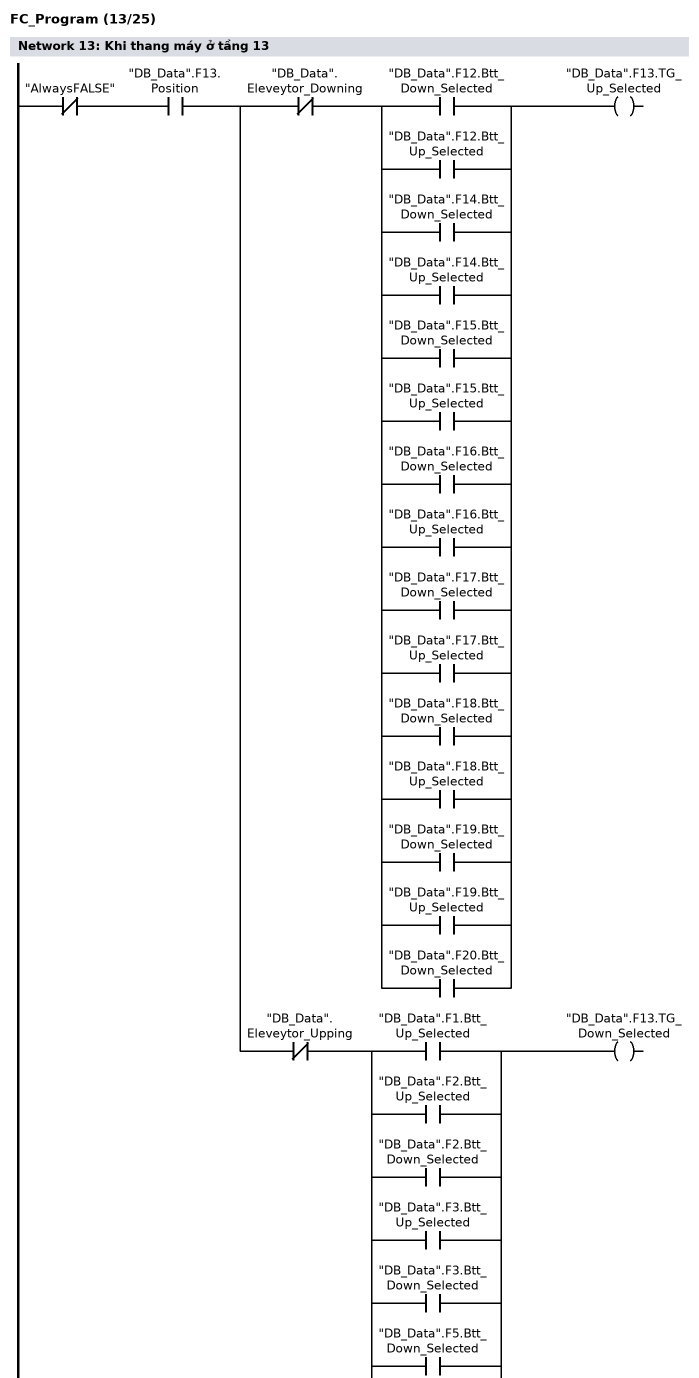
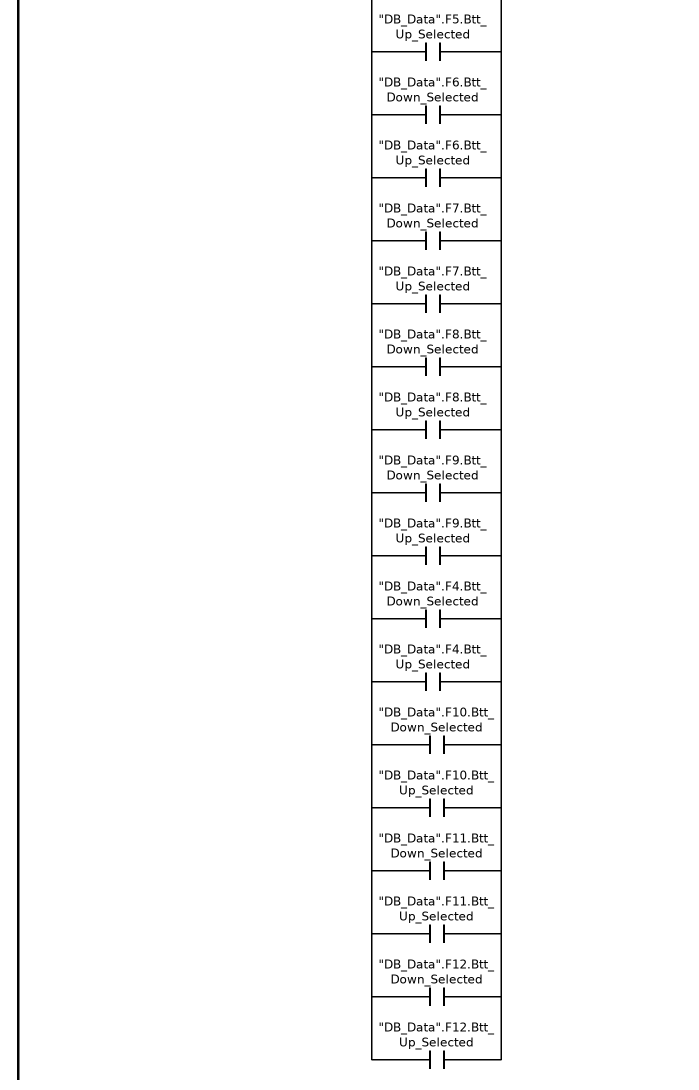
   RUNG wire#powerrail
      I_Contact( "AlwaysFALSE" )
      Contact( "DB_Data".F13.Position )
      wire#w1
      I_Contact( "DB_Data".Eleveytor_Downing )
      wire#w2
      Contact( "DB_Data".F12.Btt_Down_Selected )
      wire#w3
      Coil( "DB_Data".F13.TG_Up_Selected )
   END_RUNG
   RUNG wire#w2
      Contact( "DB_Data".F12.Btt_Up_Selected )
   END_RUNG wire#w3
   RUNG wire#w2
      Contact( "DB_Data".F14.Btt_Down_Selected )
   END_RUNG wire#w3
   RUNG wire#w2
      Contact( "DB_Data".F14.Btt_Up_Selected )
   END_RUNG wire#w3
   RUNG wire#w2
      Contact( "DB_Data".F15.Btt_Down_Selected )
   END_RUNG wire#w3
   RUNG wire#w2
      Contact( "DB_Data".F15.Btt_Up_Selected )
   END_RUNG wire#w3
   RUNG wire#w2
      Contact( "DB_Data".F16.Btt_Down_Selected )
   END_RUNG wire#w3
   RUNG wire#w2
      Contact( "DB_Data".F16.Btt_Up_Selected )
   END_RUNG wire#w3
   RUNG wire#w2
      Contact( "DB_Data".F17.Btt_Down_Selected )
   END_RUNG wire#w3
   RUNG wire#w2
      Contact( "DB_Data".F17.Btt_Up_Selected )
   END_RUNG wire#w3
   RUNG wire#w2
      Contact( "DB_Data".F18.Btt_Down_Selected )
   END_RUNG wire#w3
   RUNG wire#w2
      Contact( "DB_Data".F18.Btt_Up_Selected )
   END_RUNG wire#w3
   RUNG wire#w2
      Contact( "DB_Data".F19.Btt_Down_Selected )
   END_RUNG wire#w3
   RUNG wire#w2
      Contact( "DB_Data".F19.Btt_Up_Selected )
   END_RUNG wire#w3
   RUNG wire#w2
      Contact( "DB_Data".F20.Btt_Down_Selected )
   END_RUNG wire#w3
   RUNG wire#w1
      I_Contact( "DB_Data".Eleveytor_Upping )
      wire#w4
      Contact( "DB_Data".F1.Btt_Up_Selected )
      wire#w5
      Coil( "DB_Data".F13.TG_Down_Selected )
   END_RUNG
   RUNG wire#w4
      Contact( "DB_Data".F2.Btt_Up_Selected )
   END_RUNG wire#w5
   RUNG wire#w4
      Contact( "DB_Data".F2.Btt_Down_Selected )
   END_RUNG wire#w5
   RUNG wire#w4
      Contact( "DB_Data".F3.Btt_Up_Selected )
   END_RUNG wire#w5
   RUNG wire#w4
      Contact( "DB_Data".F3.Btt_Down_Selected )
   END_RUNG wire#w5
   RUNG wire#w4
      Contact( "DB_Data".F5.Btt_Down_Selected )
   END_RUNG wire#w5
   RUNG wire#w4
      Contact( "DB_Data".F5.Btt_Up_Selected )
   END_RUNG wire#w5
   RUNG wire#w4
      Contact( "DB_Data".F6.Btt_Down_Selected )
   END_RUNG wire#w5
   RUNG wire#w4
      Contact( "DB_Data".F6.Btt_Up_Selected )
   END_RUNG wire#w5
   RUNG wire#w4
      Contact( "DB_Data".F7.Btt_Down_Selected )
   END_RUNG wire#w5
   RUNG wire#w4
      Contact( "DB_Data".F7.Btt_Up_Selected )
   END_RUNG wire#w5
   RUNG wire#w4
      Contact( "DB_Data".F8.Btt_Down_Selected )
   END_RUNG wire#w5
   RUNG wire#w4
      Contact( "DB_Data".F8.Btt_Up_Selected )
   END_RUNG wire#w5
   RUNG wire#w4
      Contact( "DB_Data".F9.Btt_Down_Selected )
   END_RUNG wire#w5
   RUNG wire#w4
      Contact( "DB_Data".F9.Btt_Up_Selected )
   END_RUNG wire#w5
   RUNG wire#w4
      Contact( "DB_Data".F4.Btt_Down_Selected )
   END_RUNG wire#w5
   RUNG wire#w4
      Contact( "DB_Data".F4.Btt_Up_Selected )
   END_RUNG wire#w5
   RUNG wire#w4
      Contact( "DB_Data".F10.Btt_Down_Selected )
   END_RUNG wire#w5
   RUNG wire#w4
      Contact( "DB_Data".F10.Btt_Up_Selected )
   END_RUNG wire#w5
   RUNG wire#w4
      Contact( "DB_Data".F11.Btt_Down_Selected )
   END_RUNG wire#w5
   RUNG wire#w4
      Contact( "DB_Data".F11.Btt_Up_Selected )
   END_RUNG wire#w5
   RUNG wire#w4
      Contact( "DB_Data".F12.Btt_Down_Selected )
   END_RUNG wire#w5
   RUNG wire#w4
      Contact( "DB_Data".F12.Btt_Up_Selected )
   END_RUNG wire#w5
   // the same network as SCL:
   #_w1 := NOT "AlwaysFALSE" AND "DB_Data".F13.Position;
   "DB_Data".F13.TG_Up_Selected := #_w1 AND NOT "DB_Data".Eleveytor_Downing AND ("DB_Data".F12.Btt_Down_Selected OR "DB_Data".F12.Btt_Up_Selected OR "DB_Data".F14.Btt_Down_Selected OR "DB_Data".F14.Btt_Up_Selected OR "DB_Data".F15.Btt_Down_Selected OR "DB_Data".F15.Btt_Up_Selected OR "DB_Data".F16.Btt_Down_Selected OR "DB_Data".F16.Btt_Up_Selected OR "DB_Data".F17.Btt_Down_Selected OR "DB_Data".F17.Btt_Up_Selected OR "DB_Data".F18.Btt_Down_Selected OR "DB_Data".F18.Btt_Up_Selected OR "DB_Data".F19.Btt_Down_Selected OR "DB_Data".F19.Btt_Up_Selected OR "DB_Data".F20.Btt_Down_Selected);
   "DB_Data".F13.TG_Down_Selected := #_w1 AND NOT "DB_Data".Eleveytor_Upping AND ("DB_Data".F1.Btt_Up_Selected OR "DB_Data".F2.Btt_Up_Selected OR "DB_Data".F2.Btt_Down_Selected OR "DB_Data".F3.Btt_Up_Selected OR "DB_Data".F3.Btt_Down_Selected OR "DB_Data".F5.Btt_Down_Selected OR "DB_Data".F5.Btt_Up_Selected OR "DB_Data".F6.Btt_Down_Selected OR "DB_Data".F6.Btt_Up_Selected OR "DB_Data".F7.Btt_Down_Selected OR "DB_Data".F7.Btt_Up_Selected OR "DB_Data".F8.Btt_Down_Selected OR "DB_Data".F8.Btt_Up_Selected OR "DB_Data".F9.Btt_Down_Selected OR "DB_Data".F9.Btt_Up_Selected OR "DB_Data".F4.Btt_Down_Selected OR "DB_Data".F4.Btt_Up_Selected OR "DB_Data".F10.Btt_Down_Selected OR "DB_Data".F10.Btt_Up_Selected OR "DB_Data".F11.Btt_Down_Selected OR "DB_Data".F11.Btt_Up_Selected OR "DB_Data".F12.Btt_Down_Selected OR "DB_Data".F12.Btt_Up_Selected);
END_REGION

REGION Network 14: Khi thang máy ở tầng 14
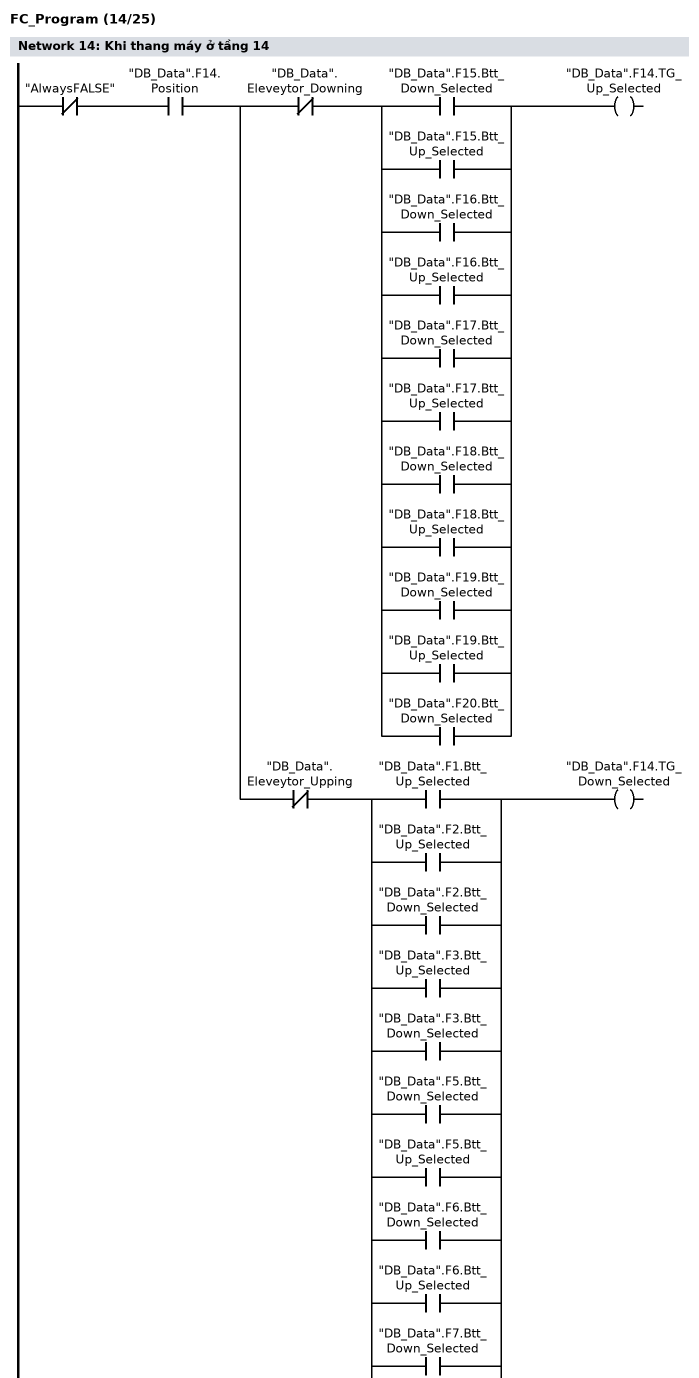
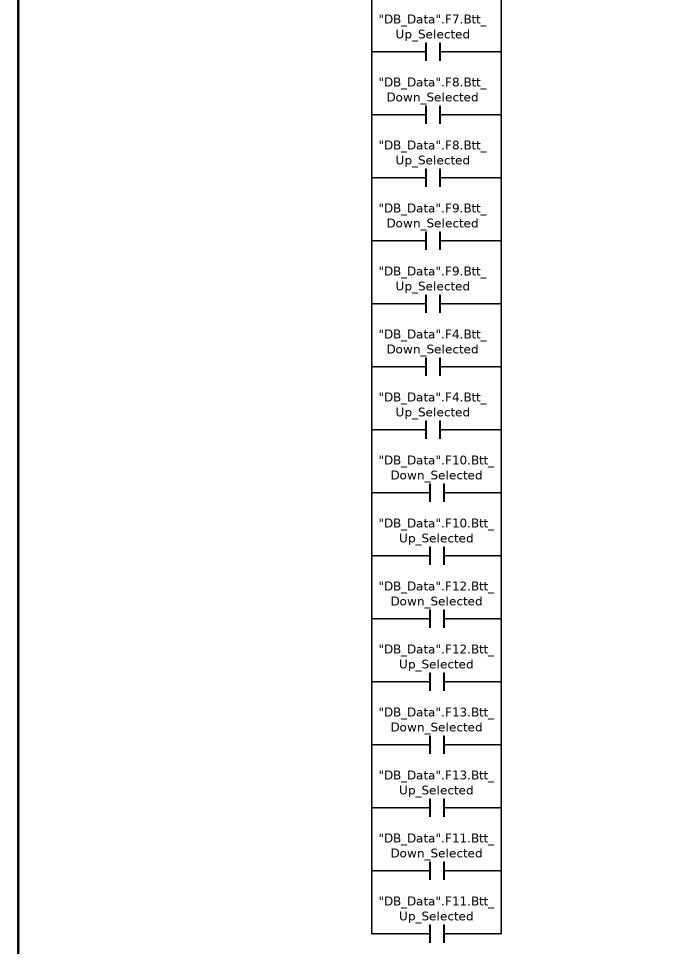
   RUNG wire#powerrail
      I_Contact( "AlwaysFALSE" )
      Contact( "DB_Data".F14.Position )
      wire#w1
      I_Contact( "DB_Data".Eleveytor_Downing )
      wire#w2
      Contact( "DB_Data".F15.Btt_Down_Selected )
      wire#w3
      Coil( "DB_Data".F14.TG_Up_Selected )
   END_RUNG
   RUNG wire#w2
      Contact( "DB_Data".F15.Btt_Up_Selected )
   END_RUNG wire#w3
   RUNG wire#w2
      Contact( "DB_Data".F16.Btt_Down_Selected )
   END_RUNG wire#w3
   RUNG wire#w2
      Contact( "DB_Data".F16.Btt_Up_Selected )
   END_RUNG wire#w3
   RUNG wire#w2
      Contact( "DB_Data".F17.Btt_Down_Selected )
   END_RUNG wire#w3
   RUNG wire#w2
      Contact( "DB_Data".F17.Btt_Up_Selected )
   END_RUNG wire#w3
   RUNG wire#w2
      Contact( "DB_Data".F18.Btt_Down_Selected )
   END_RUNG wire#w3
   RUNG wire#w2
      Contact( "DB_Data".F18.Btt_Up_Selected )
   END_RUNG wire#w3
   RUNG wire#w2
      Contact( "DB_Data".F19.Btt_Down_Selected )
   END_RUNG wire#w3
   RUNG wire#w2
      Contact( "DB_Data".F19.Btt_Up_Selected )
   END_RUNG wire#w3
   RUNG wire#w2
      Contact( "DB_Data".F20.Btt_Down_Selected )
   END_RUNG wire#w3
   RUNG wire#w1
      I_Contact( "DB_Data".Eleveytor_Upping )
      wire#w4
      Contact( "DB_Data".F1.Btt_Up_Selected )
      wire#w5
      Coil( "DB_Data".F14.TG_Down_Selected )
   END_RUNG
   RUNG wire#w4
      Contact( "DB_Data".F2.Btt_Up_Selected )
   END_RUNG wire#w5
   RUNG wire#w4
      Contact( "DB_Data".F2.Btt_Down_Selected )
   END_RUNG wire#w5
   RUNG wire#w4
      Contact( "DB_Data".F3.Btt_Up_Selected )
   END_RUNG wire#w5
   RUNG wire#w4
      Contact( "DB_Data".F3.Btt_Down_Selected )
   END_RUNG wire#w5
   RUNG wire#w4
      Contact( "DB_Data".F5.Btt_Down_Selected )
   END_RUNG wire#w5
   RUNG wire#w4
      Contact( "DB_Data".F5.Btt_Up_Selected )
   END_RUNG wire#w5
   RUNG wire#w4
      Contact( "DB_Data".F6.Btt_Down_Selected )
   END_RUNG wire#w5
   RUNG wire#w4
      Contact( "DB_Data".F6.Btt_Up_Selected )
   END_RUNG wire#w5
   RUNG wire#w4
      Contact( "DB_Data".F7.Btt_Down_Selected )
   END_RUNG wire#w5
   RUNG wire#w4
      Contact( "DB_Data".F7.Btt_Up_Selected )
   END_RUNG wire#w5
   RUNG wire#w4
      Contact( "DB_Data".F8.Btt_Down_Selected )
   END_RUNG wire#w5
   RUNG wire#w4
      Contact( "DB_Data".F8.Btt_Up_Selected )
   END_RUNG wire#w5
   RUNG wire#w4
      Contact( "DB_Data".F9.Btt_Down_Selected )
   END_RUNG wire#w5
   RUNG wire#w4
      Contact( "DB_Data".F9.Btt_Up_Selected )
   END_RUNG wire#w5
   RUNG wire#w4
      Contact( "DB_Data".F4.Btt_Down_Selected )
   END_RUNG wire#w5
   RUNG wire#w4
      Contact( "DB_Data".F4.Btt_Up_Selected )
   END_RUNG wire#w5
   RUNG wire#w4
      Contact( "DB_Data".F10.Btt_Down_Selected )
   END_RUNG wire#w5
   RUNG wire#w4
      Contact( "DB_Data".F10.Btt_Up_Selected )
   END_RUNG wire#w5
   RUNG wire#w4
      Contact( "DB_Data".F12.Btt_Down_Selected )
   END_RUNG wire#w5
   RUNG wire#w4
      Contact( "DB_Data".F12.Btt_Up_Selected )
   END_RUNG wire#w5
   RUNG wire#w4
      Contact( "DB_Data".F13.Btt_Down_Selected )
   END_RUNG wire#w5
   RUNG wire#w4
      Contact( "DB_Data".F13.Btt_Up_Selected )
   END_RUNG wire#w5
   RUNG wire#w4
      Contact( "DB_Data".F11.Btt_Down_Selected )
   END_RUNG wire#w5
   RUNG wire#w4
      Contact( "DB_Data".F11.Btt_Up_Selected )
   END_RUNG wire#w5
   // the same network as SCL:
   #_w1 := NOT "AlwaysFALSE" AND "DB_Data".F14.Position;
   "DB_Data".F14.TG_Up_Selected := #_w1 AND NOT "DB_Data".Eleveytor_Downing AND ("DB_Data".F15.Btt_Down_Selected OR "DB_Data".F15.Btt_Up_Selected OR "DB_Data".F16.Btt_Down_Selected OR "DB_Data".F16.Btt_Up_Selected OR "DB_Data".F17.Btt_Down_Selected OR "DB_Data".F17.Btt_Up_Selected OR "DB_Data".F18.Btt_Down_Selected OR "DB_Data".F18.Btt_Up_Selected OR "DB_Data".F19.Btt_Down_Selected OR "DB_Data".F19.Btt_Up_Selected OR "DB_Data".F20.Btt_Down_Selected);
   "DB_Data".F14.TG_Down_Selected := #_w1 AND NOT "DB_Data".Eleveytor_Upping AND ("DB_Data".F1.Btt_Up_Selected OR "DB_Data".F2.Btt_Up_Selected OR "DB_Data".F2.Btt_Down_Selected OR "DB_Data".F3.Btt_Up_Selected OR "DB_Data".F3.Btt_Down_Selected OR "DB_Data".F5.Btt_Down_Selected OR "DB_Data".F5.Btt_Up_Selected OR "DB_Data".F6.Btt_Down_Selected OR "DB_Data".F6.Btt_Up_Selected OR "DB_Data".F7.Btt_Down_Selected OR "DB_Data".F7.Btt_Up_Selected OR "DB_Data".F8.Btt_Down_Selected OR "DB_Data".F8.Btt_Up_Selected OR "DB_Data".F9.Btt_Down_Selected OR "DB_Data".F9.Btt_Up_Selected OR "DB_Data".F4.Btt_Down_Selected OR "DB_Data".F4.Btt_Up_Selected OR "DB_Data".F10.Btt_Down_Selected OR "DB_Data".F10.Btt_Up_Selected OR "DB_Data".F12.Btt_Down_Selected OR "DB_Data".F12.Btt_Up_Selected OR "DB_Data".F13.Btt_Down_Selected OR "DB_Data".F13.Btt_Up_Selected OR "DB_Data".F11.Btt_Down_Selected OR "DB_Data".F11.Btt_Up_Selected);
END_REGION

REGION Network 15: Khi thang máy ở tầng 15
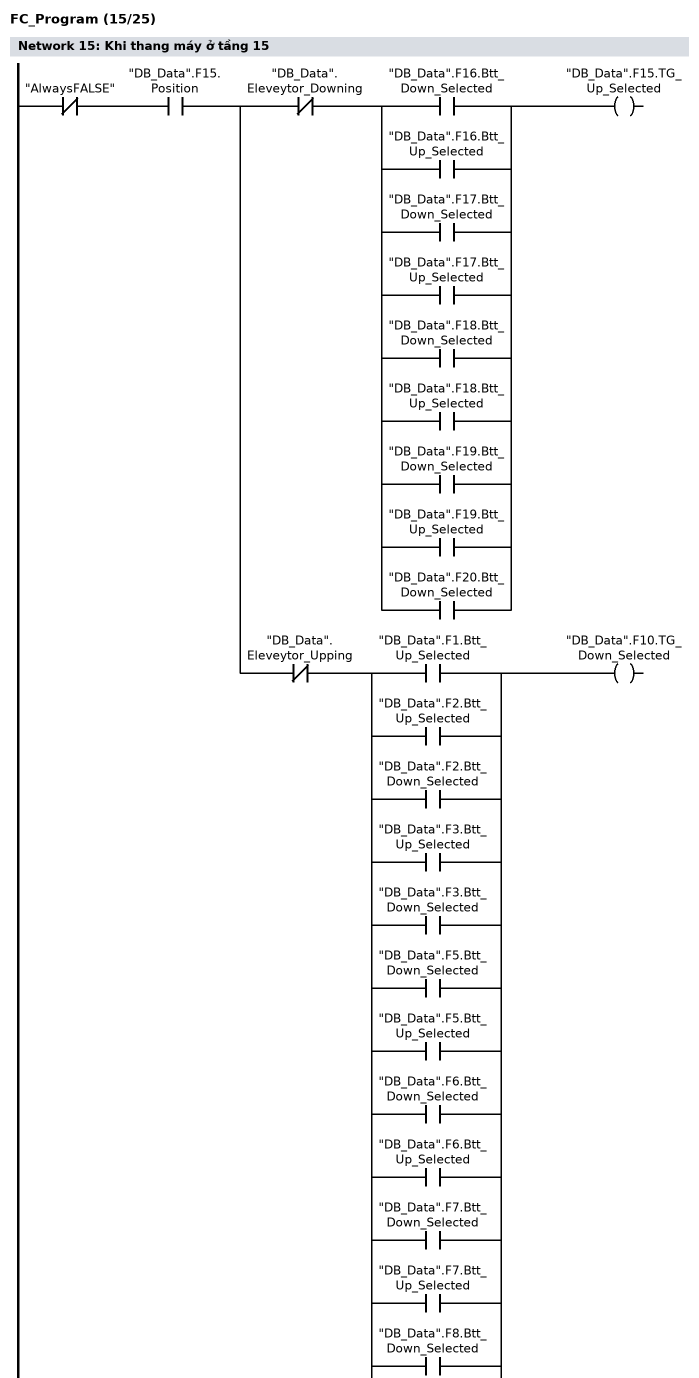
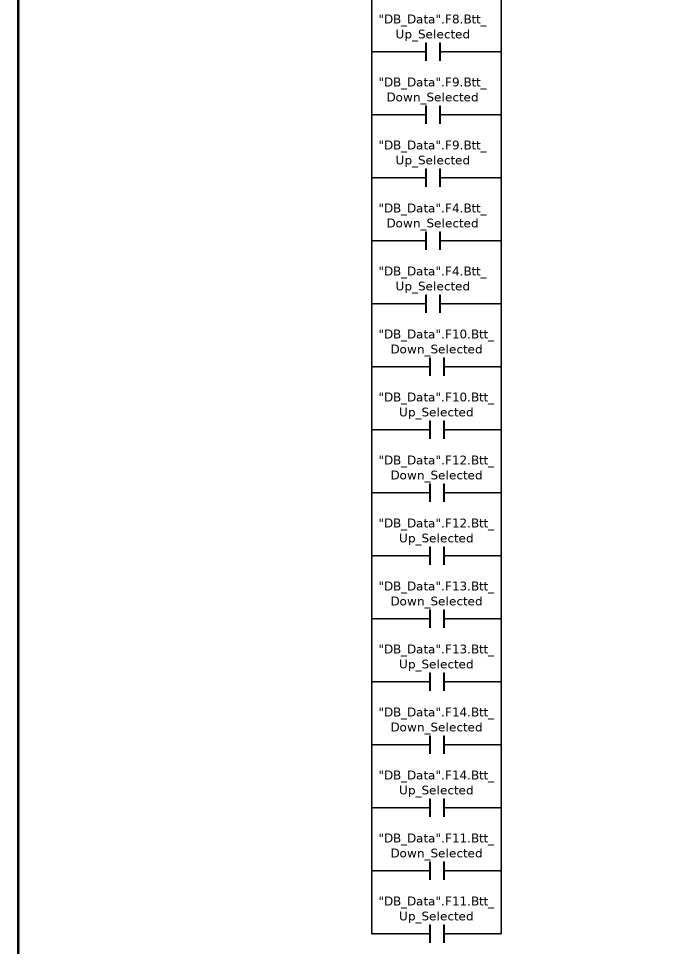
   RUNG wire#powerrail
      I_Contact( "AlwaysFALSE" )
      Contact( "DB_Data".F15.Position )
      wire#w1
      I_Contact( "DB_Data".Eleveytor_Downing )
      wire#w2
      Contact( "DB_Data".F16.Btt_Down_Selected )
      wire#w3
      Coil( "DB_Data".F15.TG_Up_Selected )
   END_RUNG
   RUNG wire#w2
      Contact( "DB_Data".F16.Btt_Up_Selected )
   END_RUNG wire#w3
   RUNG wire#w2
      Contact( "DB_Data".F17.Btt_Down_Selected )
   END_RUNG wire#w3
   RUNG wire#w2
      Contact( "DB_Data".F17.Btt_Up_Selected )
   END_RUNG wire#w3
   RUNG wire#w2
      Contact( "DB_Data".F18.Btt_Down_Selected )
   END_RUNG wire#w3
   RUNG wire#w2
      Contact( "DB_Data".F18.Btt_Up_Selected )
   END_RUNG wire#w3
   RUNG wire#w2
      Contact( "DB_Data".F19.Btt_Down_Selected )
   END_RUNG wire#w3
   RUNG wire#w2
      Contact( "DB_Data".F19.Btt_Up_Selected )
   END_RUNG wire#w3
   RUNG wire#w2
      Contact( "DB_Data".F20.Btt_Down_Selected )
   END_RUNG wire#w3
   RUNG wire#w1
      I_Contact( "DB_Data".Eleveytor_Upping )
      wire#w4
      Contact( "DB_Data".F1.Btt_Up_Selected )
      wire#w5
      Coil( "DB_Data".F10.TG_Down_Selected )
   END_RUNG
   RUNG wire#w4
      Contact( "DB_Data".F2.Btt_Up_Selected )
   END_RUNG wire#w5
   RUNG wire#w4
      Contact( "DB_Data".F2.Btt_Down_Selected )
   END_RUNG wire#w5
   RUNG wire#w4
      Contact( "DB_Data".F3.Btt_Up_Selected )
   END_RUNG wire#w5
   RUNG wire#w4
      Contact( "DB_Data".F3.Btt_Down_Selected )
   END_RUNG wire#w5
   RUNG wire#w4
      Contact( "DB_Data".F5.Btt_Down_Selected )
   END_RUNG wire#w5
   RUNG wire#w4
      Contact( "DB_Data".F5.Btt_Up_Selected )
   END_RUNG wire#w5
   RUNG wire#w4
      Contact( "DB_Data".F6.Btt_Down_Selected )
   END_RUNG wire#w5
   RUNG wire#w4
      Contact( "DB_Data".F6.Btt_Up_Selected )
   END_RUNG wire#w5
   RUNG wire#w4
      Contact( "DB_Data".F7.Btt_Down_Selected )
   END_RUNG wire#w5
   RUNG wire#w4
      Contact( "DB_Data".F7.Btt_Up_Selected )
   END_RUNG wire#w5
   RUNG wire#w4
      Contact( "DB_Data".F8.Btt_Down_Selected )
   END_RUNG wire#w5
   RUNG wire#w4
      Contact( "DB_Data".F8.Btt_Up_Selected )
   END_RUNG wire#w5
   RUNG wire#w4
      Contact( "DB_Data".F9.Btt_Down_Selected )
   END_RUNG wire#w5
   RUNG wire#w4
      Contact( "DB_Data".F9.Btt_Up_Selected )
   END_RUNG wire#w5
   RUNG wire#w4
      Contact( "DB_Data".F4.Btt_Down_Selected )
   END_RUNG wire#w5
   RUNG wire#w4
      Contact( "DB_Data".F4.Btt_Up_Selected )
   END_RUNG wire#w5
   RUNG wire#w4
      Contact( "DB_Data".F10.Btt_Down_Selected )
   END_RUNG wire#w5
   RUNG wire#w4
      Contact( "DB_Data".F10.Btt_Up_Selected )
   END_RUNG wire#w5
   RUNG wire#w4
      Contact( "DB_Data".F12.Btt_Down_Selected )
   END_RUNG wire#w5
   RUNG wire#w4
      Contact( "DB_Data".F12.Btt_Up_Selected )
   END_RUNG wire#w5
   RUNG wire#w4
      Contact( "DB_Data".F13.Btt_Down_Selected )
   END_RUNG wire#w5
   RUNG wire#w4
      Contact( "DB_Data".F13.Btt_Up_Selected )
   END_RUNG wire#w5
   RUNG wire#w4
      Contact( "DB_Data".F14.Btt_Down_Selected )
   END_RUNG wire#w5
   RUNG wire#w4
      Contact( "DB_Data".F14.Btt_Up_Selected )
   END_RUNG wire#w5
   RUNG wire#w4
      Contact( "DB_Data".F11.Btt_Down_Selected )
   END_RUNG wire#w5
   RUNG wire#w4
      Contact( "DB_Data".F11.Btt_Up_Selected )
   END_RUNG wire#w5
   // the same network as SCL:
   #_w1 := NOT "AlwaysFALSE" AND "DB_Data".F15.Position;
   "DB_Data".F15.TG_Up_Selected := #_w1 AND NOT "DB_Data".Eleveytor_Downing AND ("DB_Data".F16.Btt_Down_Selected OR "DB_Data".F16.Btt_Up_Selected OR "DB_Data".F17.Btt_Down_Selected OR "DB_Data".F17.Btt_Up_Selected OR "DB_Data".F18.Btt_Down_Selected OR "DB_Data".F18.Btt_Up_Selected OR "DB_Data".F19.Btt_Down_Selected OR "DB_Data".F19.Btt_Up_Selected OR "DB_Data".F20.Btt_Down_Selected);
   "DB_Data".F10.TG_Down_Selected := #_w1 AND NOT "DB_Data".Eleveytor_Upping AND ("DB_Data".F1.Btt_Up_Selected OR "DB_Data".F2.Btt_Up_Selected OR "DB_Data".F2.Btt_Down_Selected OR "DB_Data".F3.Btt_Up_Selected OR "DB_Data".F3.Btt_Down_Selected OR "DB_Data".F5.Btt_Down_Selected OR "DB_Data".F5.Btt_Up_Selected OR "DB_Data".F6.Btt_Down_Selected OR "DB_Data".F6.Btt_Up_Selected OR "DB_Data".F7.Btt_Down_Selected OR "DB_Data".F7.Btt_Up_Selected OR "DB_Data".F8.Btt_Down_Selected OR "DB_Data".F8.Btt_Up_Selected OR "DB_Data".F9.Btt_Down_Selected OR "DB_Data".F9.Btt_Up_Selected OR "DB_Data".F4.Btt_Down_Selected OR "DB_Data".F4.Btt_Up_Selected OR "DB_Data".F10.Btt_Down_Selected OR "DB_Data".F10.Btt_Up_Selected OR "DB_Data".F12.Btt_Down_Selected OR "DB_Data".F12.Btt_Up_Selected OR "DB_Data".F13.Btt_Down_Selected OR "DB_Data".F13.Btt_Up_Selected OR "DB_Data".F14.Btt_Down_Selected OR "DB_Data".F14.Btt_Up_Selected OR "DB_Data".F11.Btt_Down_Selected OR "DB_Data".F11.Btt_Up_Selected);
END_REGION

REGION Network 16: Khi thang máy ở tầng 16
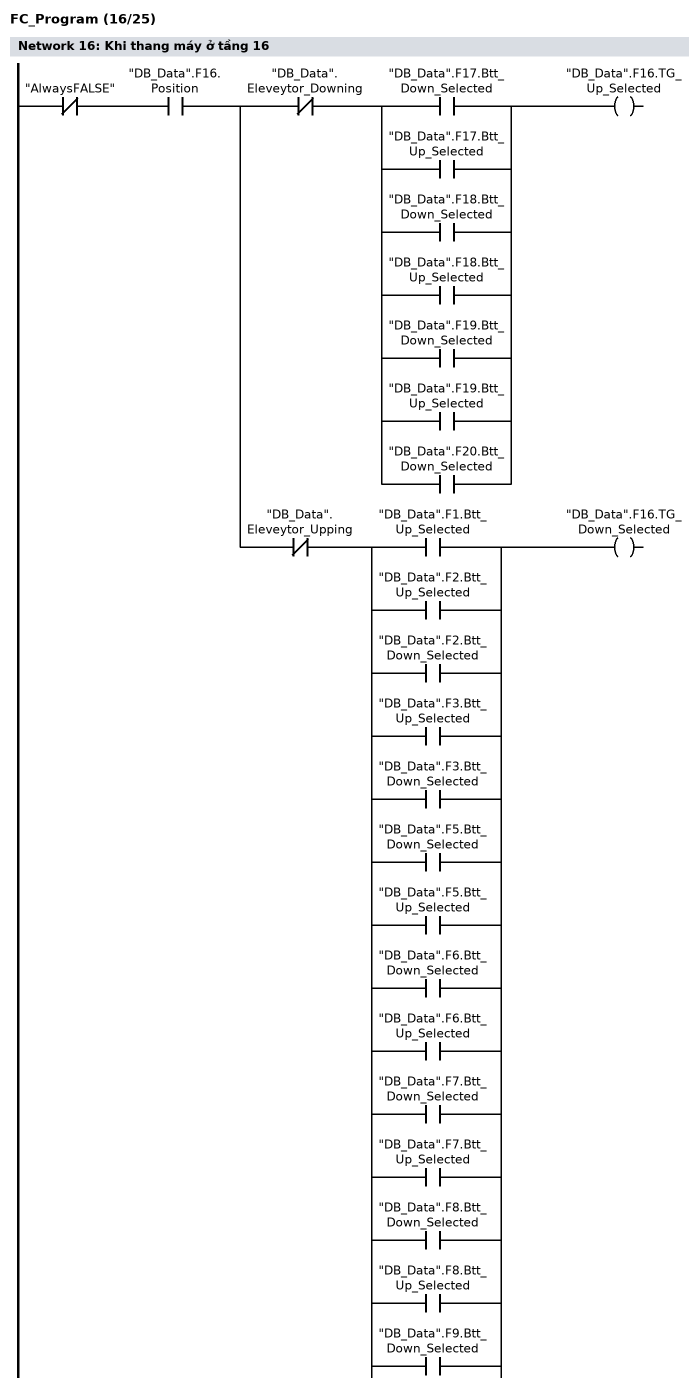
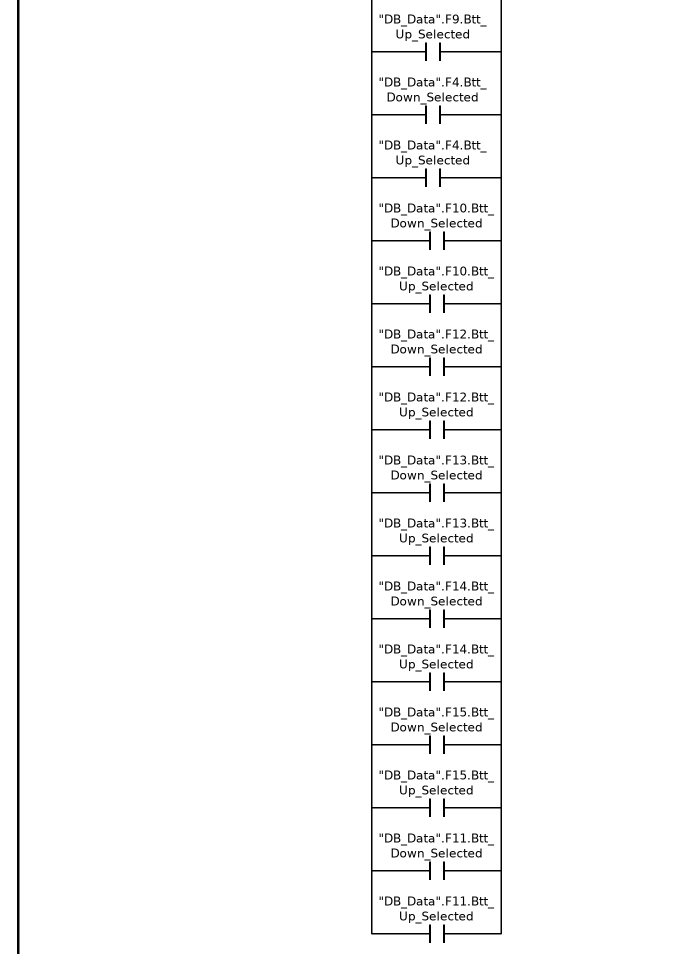
   RUNG wire#powerrail
      I_Contact( "AlwaysFALSE" )
      Contact( "DB_Data".F16.Position )
      wire#w1
      I_Contact( "DB_Data".Eleveytor_Downing )
      wire#w2
      Contact( "DB_Data".F17.Btt_Down_Selected )
      wire#w3
      Coil( "DB_Data".F16.TG_Up_Selected )
   END_RUNG
   RUNG wire#w2
      Contact( "DB_Data".F17.Btt_Up_Selected )
   END_RUNG wire#w3
   RUNG wire#w2
      Contact( "DB_Data".F18.Btt_Down_Selected )
   END_RUNG wire#w3
   RUNG wire#w2
      Contact( "DB_Data".F18.Btt_Up_Selected )
   END_RUNG wire#w3
   RUNG wire#w2
      Contact( "DB_Data".F19.Btt_Down_Selected )
   END_RUNG wire#w3
   RUNG wire#w2
      Contact( "DB_Data".F19.Btt_Up_Selected )
   END_RUNG wire#w3
   RUNG wire#w2
      Contact( "DB_Data".F20.Btt_Down_Selected )
   END_RUNG wire#w3
   RUNG wire#w1
      I_Contact( "DB_Data".Eleveytor_Upping )
      wire#w4
      Contact( "DB_Data".F1.Btt_Up_Selected )
      wire#w5
      Coil( "DB_Data".F16.TG_Down_Selected )
   END_RUNG
   RUNG wire#w4
      Contact( "DB_Data".F2.Btt_Up_Selected )
   END_RUNG wire#w5
   RUNG wire#w4
      Contact( "DB_Data".F2.Btt_Down_Selected )
   END_RUNG wire#w5
   RUNG wire#w4
      Contact( "DB_Data".F3.Btt_Up_Selected )
   END_RUNG wire#w5
   RUNG wire#w4
      Contact( "DB_Data".F3.Btt_Down_Selected )
   END_RUNG wire#w5
   RUNG wire#w4
      Contact( "DB_Data".F5.Btt_Down_Selected )
   END_RUNG wire#w5
   RUNG wire#w4
      Contact( "DB_Data".F5.Btt_Up_Selected )
   END_RUNG wire#w5
   RUNG wire#w4
      Contact( "DB_Data".F6.Btt_Down_Selected )
   END_RUNG wire#w5
   RUNG wire#w4
      Contact( "DB_Data".F6.Btt_Up_Selected )
   END_RUNG wire#w5
   RUNG wire#w4
      Contact( "DB_Data".F7.Btt_Down_Selected )
   END_RUNG wire#w5
   RUNG wire#w4
      Contact( "DB_Data".F7.Btt_Up_Selected )
   END_RUNG wire#w5
   RUNG wire#w4
      Contact( "DB_Data".F8.Btt_Down_Selected )
   END_RUNG wire#w5
   RUNG wire#w4
      Contact( "DB_Data".F8.Btt_Up_Selected )
   END_RUNG wire#w5
   RUNG wire#w4
      Contact( "DB_Data".F9.Btt_Down_Selected )
   END_RUNG wire#w5
   RUNG wire#w4
      Contact( "DB_Data".F9.Btt_Up_Selected )
   END_RUNG wire#w5
   RUNG wire#w4
      Contact( "DB_Data".F4.Btt_Down_Selected )
   END_RUNG wire#w5
   RUNG wire#w4
      Contact( "DB_Data".F4.Btt_Up_Selected )
   END_RUNG wire#w5
   RUNG wire#w4
      Contact( "DB_Data".F10.Btt_Down_Selected )
   END_RUNG wire#w5
   RUNG wire#w4
      Contact( "DB_Data".F10.Btt_Up_Selected )
   END_RUNG wire#w5
   RUNG wire#w4
      Contact( "DB_Data".F12.Btt_Down_Selected )
   END_RUNG wire#w5
   RUNG wire#w4
      Contact( "DB_Data".F12.Btt_Up_Selected )
   END_RUNG wire#w5
   RUNG wire#w4
      Contact( "DB_Data".F13.Btt_Down_Selected )
   END_RUNG wire#w5
   RUNG wire#w4
      Contact( "DB_Data".F13.Btt_Up_Selected )
   END_RUNG wire#w5
   RUNG wire#w4
      Contact( "DB_Data".F14.Btt_Down_Selected )
   END_RUNG wire#w5
   RUNG wire#w4
      Contact( "DB_Data".F14.Btt_Up_Selected )
   END_RUNG wire#w5
   RUNG wire#w4
      Contact( "DB_Data".F15.Btt_Down_Selected )
   END_RUNG wire#w5
   RUNG wire#w4
      Contact( "DB_Data".F15.Btt_Up_Selected )
   END_RUNG wire#w5
   RUNG wire#w4
      Contact( "DB_Data".F11.Btt_Down_Selected )
   END_RUNG wire#w5
   RUNG wire#w4
      Contact( "DB_Data".F11.Btt_Up_Selected )
   END_RUNG wire#w5
   // the same network as SCL:
   #_w1 := NOT "AlwaysFALSE" AND "DB_Data".F16.Position;
   "DB_Data".F16.TG_Up_Selected := #_w1 AND NOT "DB_Data".Eleveytor_Downing AND ("DB_Data".F17.Btt_Down_Selected OR "DB_Data".F17.Btt_Up_Selected OR "DB_Data".F18.Btt_Down_Selected OR "DB_Data".F18.Btt_Up_Selected OR "DB_Data".F19.Btt_Down_Selected OR "DB_Data".F19.Btt_Up_Selected OR "DB_Data".F20.Btt_Down_Selected);
   "DB_Data".F16.TG_Down_Selected := #_w1 AND NOT "DB_Data".Eleveytor_Upping AND ("DB_Data".F1.Btt_Up_Selected OR "DB_Data".F2.Btt_Up_Selected OR "DB_Data".F2.Btt_Down_Selected OR "DB_Data".F3.Btt_Up_Selected OR "DB_Data".F3.Btt_Down_Selected OR "DB_Data".F5.Btt_Down_Selected OR "DB_Data".F5.Btt_Up_Selected OR "DB_Data".F6.Btt_Down_Selected OR "DB_Data".F6.Btt_Up_Selected OR "DB_Data".F7.Btt_Down_Selected OR "DB_Data".F7.Btt_Up_Selected OR "DB_Data".F8.Btt_Down_Selected OR "DB_Data".F8.Btt_Up_Selected OR "DB_Data".F9.Btt_Down_Selected OR "DB_Data".F9.Btt_Up_Selected OR "DB_Data".F4.Btt_Down_Selected OR "DB_Data".F4.Btt_Up_Selected OR "DB_Data".F10.Btt_Down_Selected OR "DB_Data".F10.Btt_Up_Selected OR "DB_Data".F12.Btt_Down_Selected OR "DB_Data".F12.Btt_Up_Selected OR "DB_Data".F13.Btt_Down_Selected OR "DB_Data".F13.Btt_Up_Selected OR "DB_Data".F14.Btt_Down_Selected OR "DB_Data".F14.Btt_Up_Selected OR "DB_Data".F15.Btt_Down_Selected OR "DB_Data".F15.Btt_Up_Selected OR "DB_Data".F11.Btt_Down_Selected OR "DB_Data".F11.Btt_Up_Selected);
END_REGION

REGION Network 17: Khi thang máy ở tầng 17
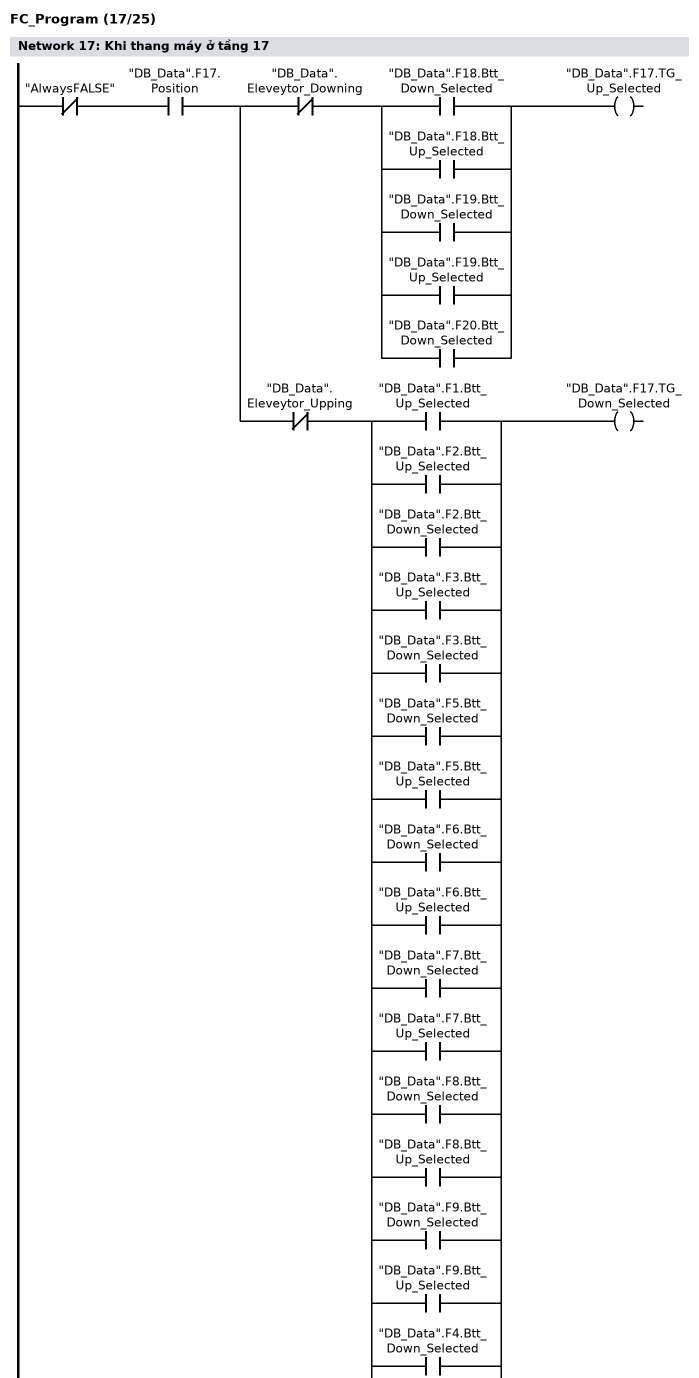
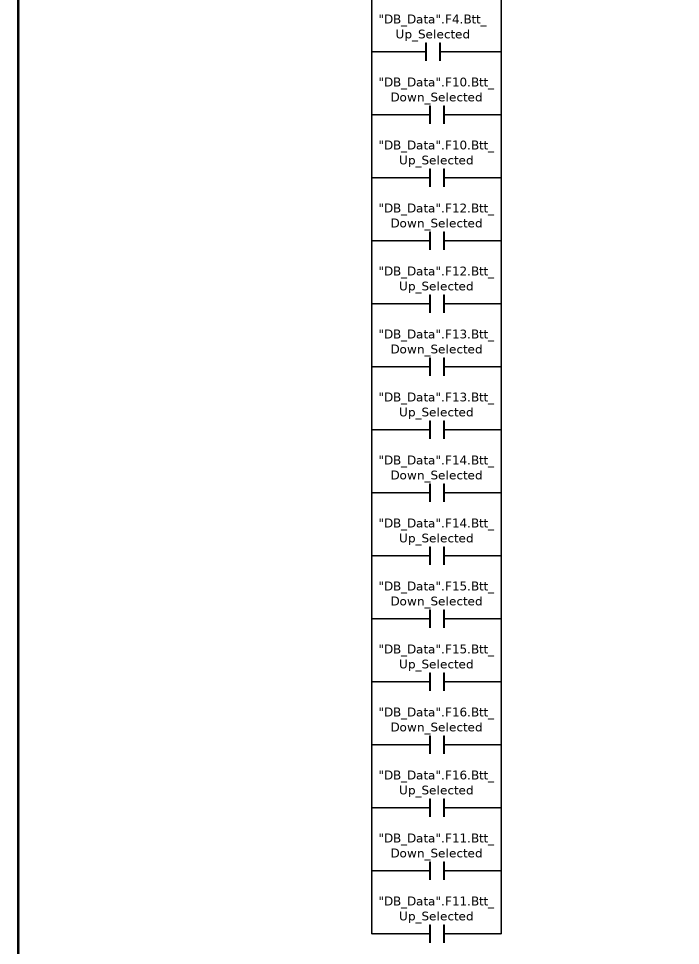
   RUNG wire#powerrail
      I_Contact( "AlwaysFALSE" )
      Contact( "DB_Data".F17.Position )
      wire#w1
      I_Contact( "DB_Data".Eleveytor_Downing )
      wire#w2
      Contact( "DB_Data".F18.Btt_Down_Selected )
      wire#w3
      Coil( "DB_Data".F17.TG_Up_Selected )
   END_RUNG
   RUNG wire#w2
      Contact( "DB_Data".F18.Btt_Up_Selected )
   END_RUNG wire#w3
   RUNG wire#w2
      Contact( "DB_Data".F19.Btt_Down_Selected )
   END_RUNG wire#w3
   RUNG wire#w2
      Contact( "DB_Data".F19.Btt_Up_Selected )
   END_RUNG wire#w3
   RUNG wire#w2
      Contact( "DB_Data".F20.Btt_Down_Selected )
   END_RUNG wire#w3
   RUNG wire#w1
      I_Contact( "DB_Data".Eleveytor_Upping )
      wire#w4
      Contact( "DB_Data".F1.Btt_Up_Selected )
      wire#w5
      Coil( "DB_Data".F17.TG_Down_Selected )
   END_RUNG
   RUNG wire#w4
      Contact( "DB_Data".F2.Btt_Up_Selected )
   END_RUNG wire#w5
   RUNG wire#w4
      Contact( "DB_Data".F2.Btt_Down_Selected )
   END_RUNG wire#w5
   RUNG wire#w4
      Contact( "DB_Data".F3.Btt_Up_Selected )
   END_RUNG wire#w5
   RUNG wire#w4
      Contact( "DB_Data".F3.Btt_Down_Selected )
   END_RUNG wire#w5
   RUNG wire#w4
      Contact( "DB_Data".F5.Btt_Down_Selected )
   END_RUNG wire#w5
   RUNG wire#w4
      Contact( "DB_Data".F5.Btt_Up_Selected )
   END_RUNG wire#w5
   RUNG wire#w4
      Contact( "DB_Data".F6.Btt_Down_Selected )
   END_RUNG wire#w5
   RUNG wire#w4
      Contact( "DB_Data".F6.Btt_Up_Selected )
   END_RUNG wire#w5
   RUNG wire#w4
      Contact( "DB_Data".F7.Btt_Down_Selected )
   END_RUNG wire#w5
   RUNG wire#w4
      Contact( "DB_Data".F7.Btt_Up_Selected )
   END_RUNG wire#w5
   RUNG wire#w4
      Contact( "DB_Data".F8.Btt_Down_Selected )
   END_RUNG wire#w5
   RUNG wire#w4
      Contact( "DB_Data".F8.Btt_Up_Selected )
   END_RUNG wire#w5
   RUNG wire#w4
      Contact( "DB_Data".F9.Btt_Down_Selected )
   END_RUNG wire#w5
   RUNG wire#w4
      Contact( "DB_Data".F9.Btt_Up_Selected )
   END_RUNG wire#w5
   RUNG wire#w4
      Contact( "DB_Data".F4.Btt_Down_Selected )
   END_RUNG wire#w5
   RUNG wire#w4
      Contact( "DB_Data".F4.Btt_Up_Selected )
   END_RUNG wire#w5
   RUNG wire#w4
      Contact( "DB_Data".F10.Btt_Down_Selected )
   END_RUNG wire#w5
   RUNG wire#w4
      Contact( "DB_Data".F10.Btt_Up_Selected )
   END_RUNG wire#w5
   RUNG wire#w4
      Contact( "DB_Data".F12.Btt_Down_Selected )
   END_RUNG wire#w5
   RUNG wire#w4
      Contact( "DB_Data".F12.Btt_Up_Selected )
   END_RUNG wire#w5
   RUNG wire#w4
      Contact( "DB_Data".F13.Btt_Down_Selected )
   END_RUNG wire#w5
   RUNG wire#w4
      Contact( "DB_Data".F13.Btt_Up_Selected )
   END_RUNG wire#w5
   RUNG wire#w4
      Contact( "DB_Data".F14.Btt_Down_Selected )
   END_RUNG wire#w5
   RUNG wire#w4
      Contact( "DB_Data".F14.Btt_Up_Selected )
   END_RUNG wire#w5
   RUNG wire#w4
      Contact( "DB_Data".F15.Btt_Down_Selected )
   END_RUNG wire#w5
   RUNG wire#w4
      Contact( "DB_Data".F15.Btt_Up_Selected )
   END_RUNG wire#w5
   RUNG wire#w4
      Contact( "DB_Data".F16.Btt_Down_Selected )
   END_RUNG wire#w5
   RUNG wire#w4
      Contact( "DB_Data".F16.Btt_Up_Selected )
   END_RUNG wire#w5
   RUNG wire#w4
      Contact( "DB_Data".F11.Btt_Down_Selected )
   END_RUNG wire#w5
   RUNG wire#w4
      Contact( "DB_Data".F11.Btt_Up_Selected )
   END_RUNG wire#w5
   // the same network as SCL:
   #_w1 := NOT "AlwaysFALSE" AND "DB_Data".F17.Position;
   "DB_Data".F17.TG_Up_Selected := #_w1 AND NOT "DB_Data".Eleveytor_Downing AND ("DB_Data".F18.Btt_Down_Selected OR "DB_Data".F18.Btt_Up_Selected OR "DB_Data".F19.Btt_Down_Selected OR "DB_Data".F19.Btt_Up_Selected OR "DB_Data".F20.Btt_Down_Selected);
   "DB_Data".F17.TG_Down_Selected := #_w1 AND NOT "DB_Data".Eleveytor_Upping AND ("DB_Data".F1.Btt_Up_Selected OR "DB_Data".F2.Btt_Up_Selected OR "DB_Data".F2.Btt_Down_Selected OR "DB_Data".F3.Btt_Up_Selected OR "DB_Data".F3.Btt_Down_Selected OR "DB_Data".F5.Btt_Down_Selected OR "DB_Data".F5.Btt_Up_Selected OR "DB_Data".F6.Btt_Down_Selected OR "DB_Data".F6.Btt_Up_Selected OR "DB_Data".F7.Btt_Down_Selected OR "DB_Data".F7.Btt_Up_Selected OR "DB_Data".F8.Btt_Down_Selected OR "DB_Data".F8.Btt_Up_Selected OR "DB_Data".F9.Btt_Down_Selected OR "DB_Data".F9.Btt_Up_Selected OR "DB_Data".F4.Btt_Down_Selected OR "DB_Data".F4.Btt_Up_Selected OR "DB_Data".F10.Btt_Down_Selected OR "DB_Data".F10.Btt_Up_Selected OR "DB_Data".F12.Btt_Down_Selected OR "DB_Data".F12.Btt_Up_Selected OR "DB_Data".F13.Btt_Down_Selected OR "DB_Data".F13.Btt_Up_Selected OR "DB_Data".F14.Btt_Down_Selected OR "DB_Data".F14.Btt_Up_Selected OR "DB_Data".F15.Btt_Down_Selected OR "DB_Data".F15.Btt_Up_Selected OR "DB_Data".F16.Btt_Down_Selected OR "DB_Data".F16.Btt_Up_Selected OR "DB_Data".F11.Btt_Down_Selected OR "DB_Data".F11.Btt_Up_Selected);
END_REGION

REGION Network 18: Khi thang máy ở tầng 18
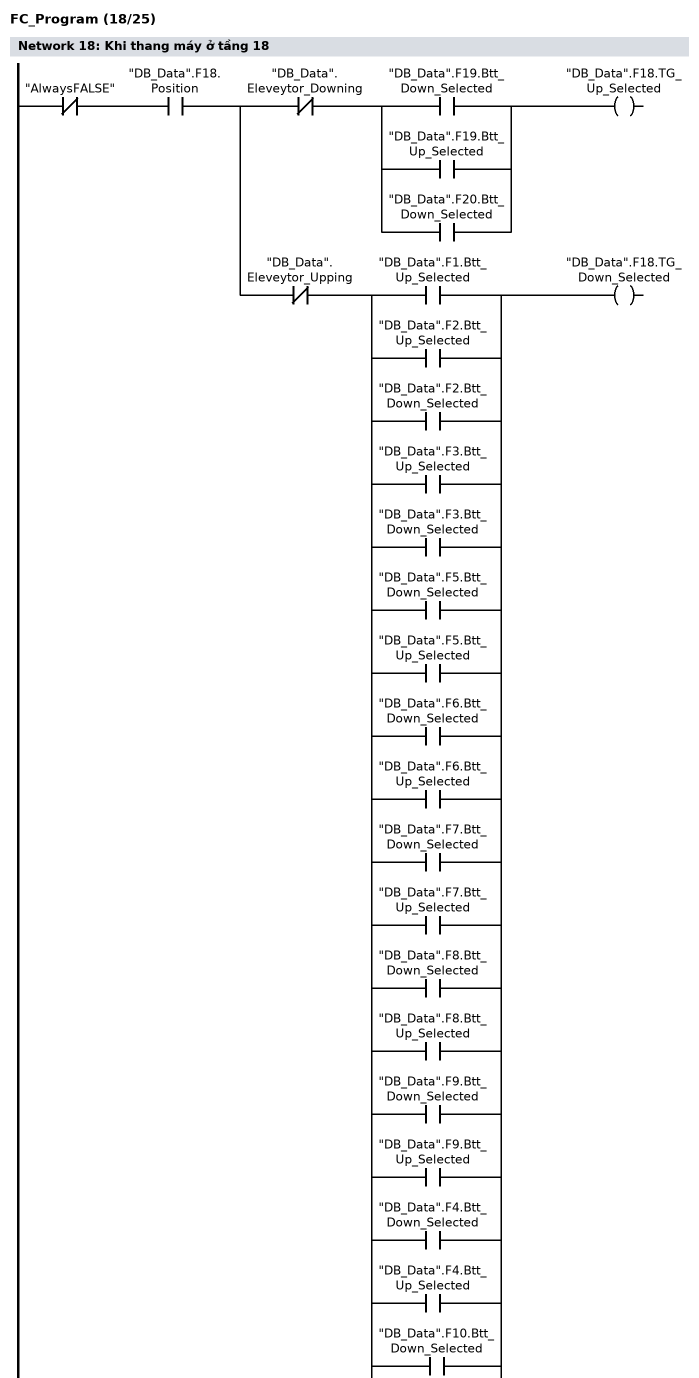
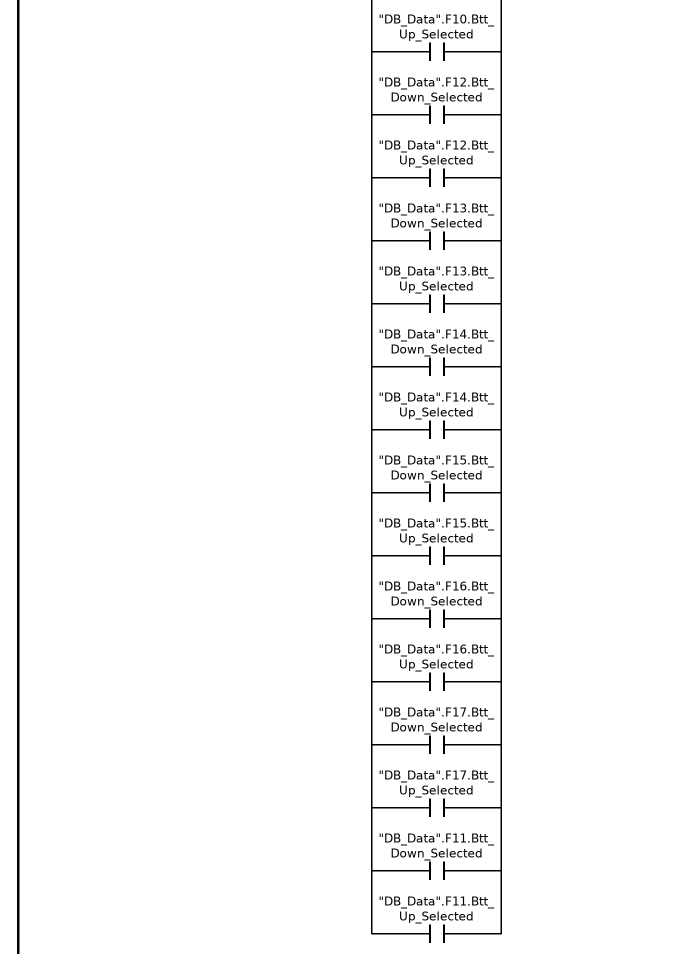
   RUNG wire#powerrail
      I_Contact( "AlwaysFALSE" )
      Contact( "DB_Data".F18.Position )
      wire#w1
      I_Contact( "DB_Data".Eleveytor_Downing )
      wire#w2
      Contact( "DB_Data".F19.Btt_Down_Selected )
      wire#w3
      Coil( "DB_Data".F18.TG_Up_Selected )
   END_RUNG
   RUNG wire#w2
      Contact( "DB_Data".F19.Btt_Up_Selected )
   END_RUNG wire#w3
   RUNG wire#w2
      Contact( "DB_Data".F20.Btt_Down_Selected )
   END_RUNG wire#w3
   RUNG wire#w1
      I_Contact( "DB_Data".Eleveytor_Upping )
      wire#w4
      Contact( "DB_Data".F1.Btt_Up_Selected )
      wire#w5
      Coil( "DB_Data".F18.TG_Down_Selected )
   END_RUNG
   RUNG wire#w4
      Contact( "DB_Data".F2.Btt_Up_Selected )
   END_RUNG wire#w5
   RUNG wire#w4
      Contact( "DB_Data".F2.Btt_Down_Selected )
   END_RUNG wire#w5
   RUNG wire#w4
      Contact( "DB_Data".F3.Btt_Up_Selected )
   END_RUNG wire#w5
   RUNG wire#w4
      Contact( "DB_Data".F3.Btt_Down_Selected )
   END_RUNG wire#w5
   RUNG wire#w4
      Contact( "DB_Data".F5.Btt_Down_Selected )
   END_RUNG wire#w5
   RUNG wire#w4
      Contact( "DB_Data".F5.Btt_Up_Selected )
   END_RUNG wire#w5
   RUNG wire#w4
      Contact( "DB_Data".F6.Btt_Down_Selected )
   END_RUNG wire#w5
   RUNG wire#w4
      Contact( "DB_Data".F6.Btt_Up_Selected )
   END_RUNG wire#w5
   RUNG wire#w4
      Contact( "DB_Data".F7.Btt_Down_Selected )
   END_RUNG wire#w5
   RUNG wire#w4
      Contact( "DB_Data".F7.Btt_Up_Selected )
   END_RUNG wire#w5
   RUNG wire#w4
      Contact( "DB_Data".F8.Btt_Down_Selected )
   END_RUNG wire#w5
   RUNG wire#w4
      Contact( "DB_Data".F8.Btt_Up_Selected )
   END_RUNG wire#w5
   RUNG wire#w4
      Contact( "DB_Data".F9.Btt_Down_Selected )
   END_RUNG wire#w5
   RUNG wire#w4
      Contact( "DB_Data".F9.Btt_Up_Selected )
   END_RUNG wire#w5
   RUNG wire#w4
      Contact( "DB_Data".F4.Btt_Down_Selected )
   END_RUNG wire#w5
   RUNG wire#w4
      Contact( "DB_Data".F4.Btt_Up_Selected )
   END_RUNG wire#w5
   RUNG wire#w4
      Contact( "DB_Data".F10.Btt_Down_Selected )
   END_RUNG wire#w5
   RUNG wire#w4
      Contact( "DB_Data".F10.Btt_Up_Selected )
   END_RUNG wire#w5
   RUNG wire#w4
      Contact( "DB_Data".F12.Btt_Down_Selected )
   END_RUNG wire#w5
   RUNG wire#w4
      Contact( "DB_Data".F12.Btt_Up_Selected )
   END_RUNG wire#w5
   RUNG wire#w4
      Contact( "DB_Data".F13.Btt_Down_Selected )
   END_RUNG wire#w5
   RUNG wire#w4
      Contact( "DB_Data".F13.Btt_Up_Selected )
   END_RUNG wire#w5
   RUNG wire#w4
      Contact( "DB_Data".F14.Btt_Down_Selected )
   END_RUNG wire#w5
   RUNG wire#w4
      Contact( "DB_Data".F14.Btt_Up_Selected )
   END_RUNG wire#w5
   RUNG wire#w4
      Contact( "DB_Data".F15.Btt_Down_Selected )
   END_RUNG wire#w5
   RUNG wire#w4
      Contact( "DB_Data".F15.Btt_Up_Selected )
   END_RUNG wire#w5
   RUNG wire#w4
      Contact( "DB_Data".F16.Btt_Down_Selected )
   END_RUNG wire#w5
   RUNG wire#w4
      Contact( "DB_Data".F16.Btt_Up_Selected )
   END_RUNG wire#w5
   RUNG wire#w4
      Contact( "DB_Data".F17.Btt_Down_Selected )
   END_RUNG wire#w5
   RUNG wire#w4
      Contact( "DB_Data".F17.Btt_Up_Selected )
   END_RUNG wire#w5
   RUNG wire#w4
      Contact( "DB_Data".F11.Btt_Down_Selected )
   END_RUNG wire#w5
   RUNG wire#w4
      Contact( "DB_Data".F11.Btt_Up_Selected )
   END_RUNG wire#w5
   // the same network as SCL:
   #_w1 := NOT "AlwaysFALSE" AND "DB_Data".F18.Position;
   "DB_Data".F18.TG_Up_Selected := #_w1 AND NOT "DB_Data".Eleveytor_Downing AND ("DB_Data".F19.Btt_Down_Selected OR "DB_Data".F19.Btt_Up_Selected OR "DB_Data".F20.Btt_Down_Selected);
   "DB_Data".F18.TG_Down_Selected := #_w1 AND NOT "DB_Data".Eleveytor_Upping AND ("DB_Data".F1.Btt_Up_Selected OR "DB_Data".F2.Btt_Up_Selected OR "DB_Data".F2.Btt_Down_Selected OR "DB_Data".F3.Btt_Up_Selected OR "DB_Data".F3.Btt_Down_Selected OR "DB_Data".F5.Btt_Down_Selected OR "DB_Data".F5.Btt_Up_Selected OR "DB_Data".F6.Btt_Down_Selected OR "DB_Data".F6.Btt_Up_Selected OR "DB_Data".F7.Btt_Down_Selected OR "DB_Data".F7.Btt_Up_Selected OR "DB_Data".F8.Btt_Down_Selected OR "DB_Data".F8.Btt_Up_Selected OR "DB_Data".F9.Btt_Down_Selected OR "DB_Data".F9.Btt_Up_Selected OR "DB_Data".F4.Btt_Down_Selected OR "DB_Data".F4.Btt_Up_Selected OR "DB_Data".F10.Btt_Down_Selected OR "DB_Data".F10.Btt_Up_Selected OR "DB_Data".F12.Btt_Down_Selected OR "DB_Data".F12.Btt_Up_Selected OR "DB_Data".F13.Btt_Down_Selected OR "DB_Data".F13.Btt_Up_Selected OR "DB_Data".F14.Btt_Down_Selected OR "DB_Data".F14.Btt_Up_Selected OR "DB_Data".F15.Btt_Down_Selected OR "DB_Data".F15.Btt_Up_Selected OR "DB_Data".F16.Btt_Down_Selected OR "DB_Data".F16.Btt_Up_Selected OR "DB_Data".F17.Btt_Down_Selected OR "DB_Data".F17.Btt_Up_Selected OR "DB_Data".F11.Btt_Down_Selected OR "DB_Data".F11.Btt_Up_Selected);
END_REGION

REGION Network 19: Khi thang máy ở tầng 19
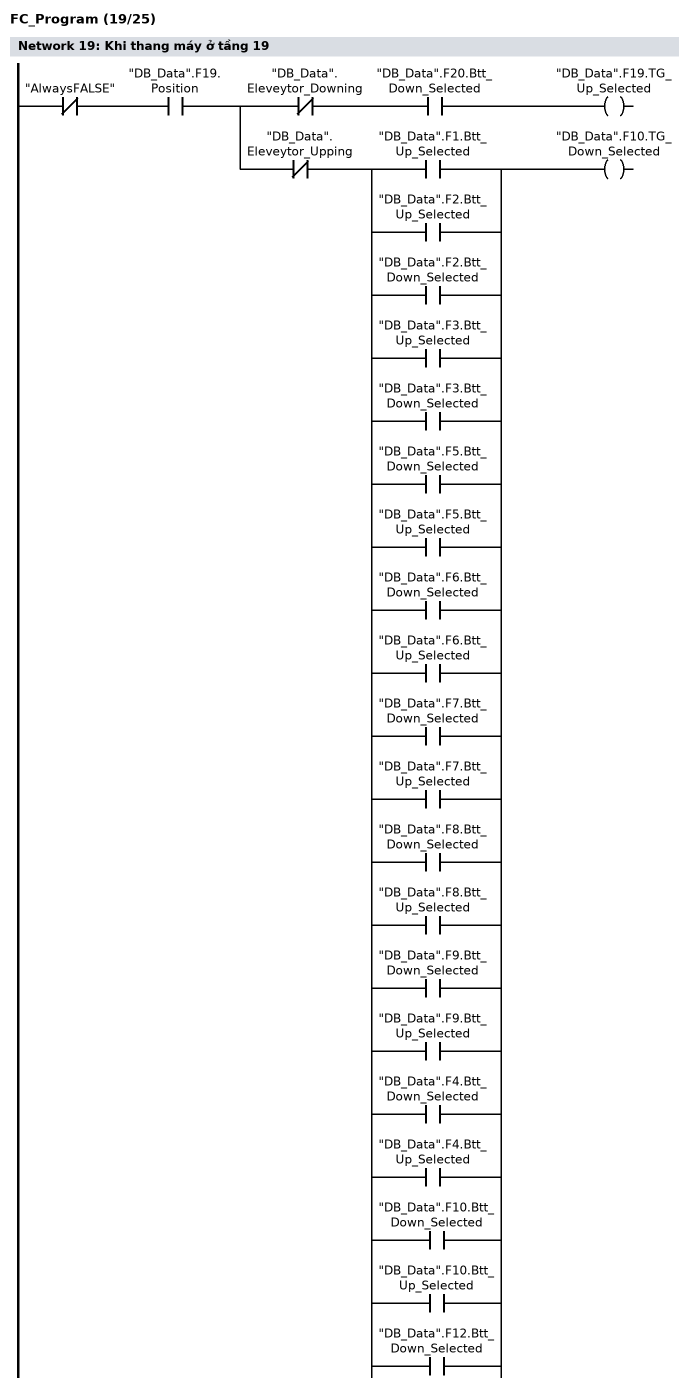
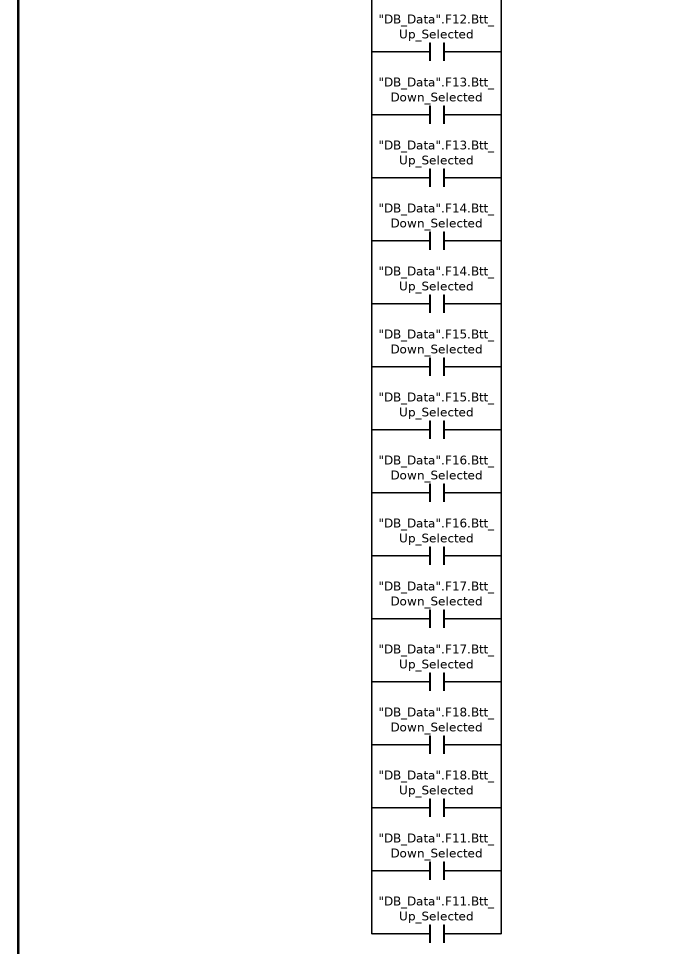
   RUNG wire#powerrail
      I_Contact( "AlwaysFALSE" )
      Contact( "DB_Data".F19.Position )
      wire#w1
      I_Contact( "DB_Data".Eleveytor_Downing )
      Contact( "DB_Data".F20.Btt_Down_Selected )
      Coil( "DB_Data".F19.TG_Up_Selected )
   END_RUNG
   RUNG wire#w1
      I_Contact( "DB_Data".Eleveytor_Upping )
      wire#w2
      Contact( "DB_Data".F1.Btt_Up_Selected )
      wire#w3
      Coil( "DB_Data".F10.TG_Down_Selected )
   END_RUNG
   RUNG wire#w2
      Contact( "DB_Data".F2.Btt_Up_Selected )
   END_RUNG wire#w3
   RUNG wire#w2
      Contact( "DB_Data".F2.Btt_Down_Selected )
   END_RUNG wire#w3
   RUNG wire#w2
      Contact( "DB_Data".F3.Btt_Up_Selected )
   END_RUNG wire#w3
   RUNG wire#w2
      Contact( "DB_Data".F3.Btt_Down_Selected )
   END_RUNG wire#w3
   RUNG wire#w2
      Contact( "DB_Data".F5.Btt_Down_Selected )
   END_RUNG wire#w3
   RUNG wire#w2
      Contact( "DB_Data".F5.Btt_Up_Selected )
   END_RUNG wire#w3
   RUNG wire#w2
      Contact( "DB_Data".F6.Btt_Down_Selected )
   END_RUNG wire#w3
   RUNG wire#w2
      Contact( "DB_Data".F6.Btt_Up_Selected )
   END_RUNG wire#w3
   RUNG wire#w2
      Contact( "DB_Data".F7.Btt_Down_Selected )
   END_RUNG wire#w3
   RUNG wire#w2
      Contact( "DB_Data".F7.Btt_Up_Selected )
   END_RUNG wire#w3
   RUNG wire#w2
      Contact( "DB_Data".F8.Btt_Down_Selected )
   END_RUNG wire#w3
   RUNG wire#w2
      Contact( "DB_Data".F8.Btt_Up_Selected )
   END_RUNG wire#w3
   RUNG wire#w2
      Contact( "DB_Data".F9.Btt_Down_Selected )
   END_RUNG wire#w3
   RUNG wire#w2
      Contact( "DB_Data".F9.Btt_Up_Selected )
   END_RUNG wire#w3
   RUNG wire#w2
      Contact( "DB_Data".F4.Btt_Down_Selected )
   END_RUNG wire#w3
   RUNG wire#w2
      Contact( "DB_Data".F4.Btt_Up_Selected )
   END_RUNG wire#w3
   RUNG wire#w2
      Contact( "DB_Data".F10.Btt_Down_Selected )
   END_RUNG wire#w3
   RUNG wire#w2
      Contact( "DB_Data".F10.Btt_Up_Selected )
   END_RUNG wire#w3
   RUNG wire#w2
      Contact( "DB_Data".F12.Btt_Down_Selected )
   END_RUNG wire#w3
   RUNG wire#w2
      Contact( "DB_Data".F12.Btt_Up_Selected )
   END_RUNG wire#w3
   RUNG wire#w2
      Contact( "DB_Data".F13.Btt_Down_Selected )
   END_RUNG wire#w3
   RUNG wire#w2
      Contact( "DB_Data".F13.Btt_Up_Selected )
   END_RUNG wire#w3
   RUNG wire#w2
      Contact( "DB_Data".F14.Btt_Down_Selected )
   END_RUNG wire#w3
   RUNG wire#w2
      Contact( "DB_Data".F14.Btt_Up_Selected )
   END_RUNG wire#w3
   RUNG wire#w2
      Contact( "DB_Data".F15.Btt_Down_Selected )
   END_RUNG wire#w3
   RUNG wire#w2
      Contact( "DB_Data".F15.Btt_Up_Selected )
   END_RUNG wire#w3
   RUNG wire#w2
      Contact( "DB_Data".F16.Btt_Down_Selected )
   END_RUNG wire#w3
   RUNG wire#w2
      Contact( "DB_Data".F16.Btt_Up_Selected )
   END_RUNG wire#w3
   RUNG wire#w2
      Contact( "DB_Data".F17.Btt_Down_Selected )
   END_RUNG wire#w3
   RUNG wire#w2
      Contact( "DB_Data".F17.Btt_Up_Selected )
   END_RUNG wire#w3
   RUNG wire#w2
      Contact( "DB_Data".F18.Btt_Down_Selected )
   END_RUNG wire#w3
   RUNG wire#w2
      Contact( "DB_Data".F18.Btt_Up_Selected )
   END_RUNG wire#w3
   RUNG wire#w2
      Contact( "DB_Data".F11.Btt_Down_Selected )
   END_RUNG wire#w3
   RUNG wire#w2
      Contact( "DB_Data".F11.Btt_Up_Selected )
   END_RUNG wire#w3
   // the same network as SCL:
   #_w1 := NOT "AlwaysFALSE" AND "DB_Data".F19.Position;
   "DB_Data".F19.TG_Up_Selected := #_w1 AND NOT "DB_Data".Eleveytor_Downing AND "DB_Data".F20.Btt_Down_Selected;
   "DB_Data".F10.TG_Down_Selected := #_w1 AND NOT "DB_Data".Eleveytor_Upping AND ("DB_Data".F1.Btt_Up_Selected OR "DB_Data".F2.Btt_Up_Selected OR "DB_Data".F2.Btt_Down_Selected OR "DB_Data".F3.Btt_Up_Selected OR "DB_Data".F3.Btt_Down_Selected OR "DB_Data".F5.Btt_Down_Selected OR "DB_Data".F5.Btt_Up_Selected OR "DB_Data".F6.Btt_Down_Selected OR "DB_Data".F6.Btt_Up_Selected OR "DB_Data".F7.Btt_Down_Selected OR "DB_Data".F7.Btt_Up_Selected OR "DB_Data".F8.Btt_Down_Selected OR "DB_Data".F8.Btt_Up_Selected OR "DB_Data".F9.Btt_Down_Selected OR "DB_Data".F9.Btt_Up_Selected OR "DB_Data".F4.Btt_Down_Selected OR "DB_Data".F4.Btt_Up_Selected OR "DB_Data".F10.Btt_Down_Selected OR "DB_Data".F10.Btt_Up_Selected OR "DB_Data".F12.Btt_Down_Selected OR "DB_Data".F12.Btt_Up_Selected OR "DB_Data".F13.Btt_Down_Selected OR "DB_Data".F13.Btt_Up_Selected OR "DB_Data".F14.Btt_Down_Selected OR "DB_Data".F14.Btt_Up_Selected OR "DB_Data".F15.Btt_Down_Selected OR "DB_Data".F15.Btt_Up_Selected OR "DB_Data".F16.Btt_Down_Selected OR "DB_Data".F16.Btt_Up_Selected OR "DB_Data".F17.Btt_Down_Selected OR "DB_Data".F17.Btt_Up_Selected OR "DB_Data".F18.Btt_Down_Selected OR "DB_Data".F18.Btt_Up_Selected OR "DB_Data".F11.Btt_Down_Selected OR "DB_Data".F11.Btt_Up_Selected);
END_REGION

REGION Network 20: Khi thang máy ở tầng 20
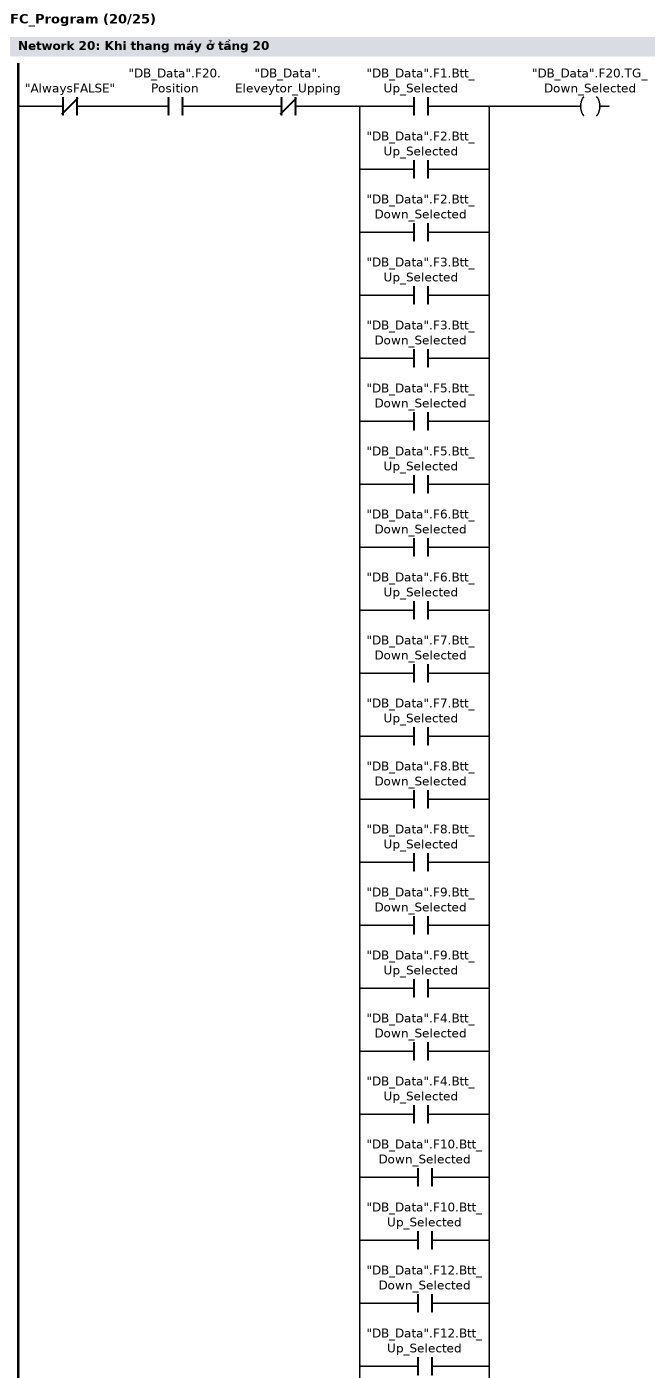
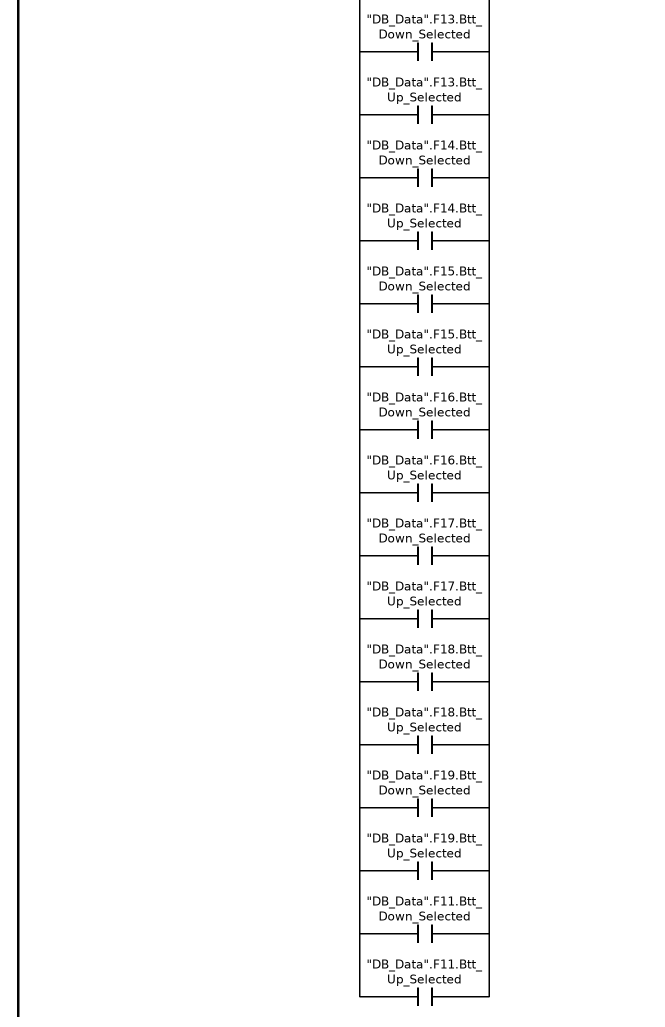
   RUNG wire#powerrail
      I_Contact( "AlwaysFALSE" )
      Contact( "DB_Data".F20.Position )
      I_Contact( "DB_Data".Eleveytor_Upping )
      wire#w1
      Contact( "DB_Data".F1.Btt_Up_Selected )
      wire#w2
      Coil( "DB_Data".F20.TG_Down_Selected )
   END_RUNG
   RUNG wire#w1
      Contact( "DB_Data".F2.Btt_Up_Selected )
   END_RUNG wire#w2
   RUNG wire#w1
      Contact( "DB_Data".F2.Btt_Down_Selected )
   END_RUNG wire#w2
   RUNG wire#w1
      Contact( "DB_Data".F3.Btt_Up_Selected )
   END_RUNG wire#w2
   RUNG wire#w1
      Contact( "DB_Data".F3.Btt_Down_Selected )
   END_RUNG wire#w2
   RUNG wire#w1
      Contact( "DB_Data".F5.Btt_Down_Selected )
   END_RUNG wire#w2
   RUNG wire#w1
      Contact( "DB_Data".F5.Btt_Up_Selected )
   END_RUNG wire#w2
   RUNG wire#w1
      Contact( "DB_Data".F6.Btt_Down_Selected )
   END_RUNG wire#w2
   RUNG wire#w1
      Contact( "DB_Data".F6.Btt_Up_Selected )
   END_RUNG wire#w2
   RUNG wire#w1
      Contact( "DB_Data".F7.Btt_Down_Selected )
   END_RUNG wire#w2
   RUNG wire#w1
      Contact( "DB_Data".F7.Btt_Up_Selected )
   END_RUNG wire#w2
   RUNG wire#w1
      Contact( "DB_Data".F8.Btt_Down_Selected )
   END_RUNG wire#w2
   RUNG wire#w1
      Contact( "DB_Data".F8.Btt_Up_Selected )
   END_RUNG wire#w2
   RUNG wire#w1
      Contact( "DB_Data".F9.Btt_Down_Selected )
   END_RUNG wire#w2
   RUNG wire#w1
      Contact( "DB_Data".F9.Btt_Up_Selected )
   END_RUNG wire#w2
   RUNG wire#w1
      Contact( "DB_Data".F4.Btt_Down_Selected )
   END_RUNG wire#w2
   RUNG wire#w1
      Contact( "DB_Data".F4.Btt_Up_Selected )
   END_RUNG wire#w2
   RUNG wire#w1
      Contact( "DB_Data".F10.Btt_Down_Selected )
   END_RUNG wire#w2
   RUNG wire#w1
      Contact( "DB_Data".F10.Btt_Up_Selected )
   END_RUNG wire#w2
   RUNG wire#w1
      Contact( "DB_Data".F12.Btt_Down_Selected )
   END_RUNG wire#w2
   RUNG wire#w1
      Contact( "DB_Data".F12.Btt_Up_Selected )
   END_RUNG wire#w2
   RUNG wire#w1
      Contact( "DB_Data".F13.Btt_Down_Selected )
   END_RUNG wire#w2
   RUNG wire#w1
      Contact( "DB_Data".F13.Btt_Up_Selected )
   END_RUNG wire#w2
   RUNG wire#w1
      Contact( "DB_Data".F14.Btt_Down_Selected )
   END_RUNG wire#w2
   RUNG wire#w1
      Contact( "DB_Data".F14.Btt_Up_Selected )
   END_RUNG wire#w2
   RUNG wire#w1
      Contact( "DB_Data".F15.Btt_Down_Selected )
   END_RUNG wire#w2
   RUNG wire#w1
      Contact( "DB_Data".F15.Btt_Up_Selected )
   END_RUNG wire#w2
   RUNG wire#w1
      Contact( "DB_Data".F16.Btt_Down_Selected )
   END_RUNG wire#w2
   RUNG wire#w1
      Contact( "DB_Data".F16.Btt_Up_Selected )
   END_RUNG wire#w2
   RUNG wire#w1
      Contact( "DB_Data".F17.Btt_Down_Selected )
   END_RUNG wire#w2
   RUNG wire#w1
      Contact( "DB_Data".F17.Btt_Up_Selected )
   END_RUNG wire#w2
   RUNG wire#w1
      Contact( "DB_Data".F18.Btt_Down_Selected )
   END_RUNG wire#w2
   RUNG wire#w1
      Contact( "DB_Data".F18.Btt_Up_Selected )
   END_RUNG wire#w2
   RUNG wire#w1
      Contact( "DB_Data".F19.Btt_Down_Selected )
   END_RUNG wire#w2
   RUNG wire#w1
      Contact( "DB_Data".F19.Btt_Up_Selected )
   END_RUNG wire#w2
   RUNG wire#w1
      Contact( "DB_Data".F11.Btt_Down_Selected )
   END_RUNG wire#w2
   RUNG wire#w1
      Contact( "DB_Data".F11.Btt_Up_Selected )
   END_RUNG wire#w2
   // the same network as SCL:
   "DB_Data".F20.TG_Down_Selected := NOT "AlwaysFALSE" AND "DB_Data".F20.Position AND NOT "DB_Data".Eleveytor_Upping AND ("DB_Data".F1.Btt_Up_Selected OR "DB_Data".F2.Btt_Up_Selected OR "DB_Data".F2.Btt_Down_Selected OR "DB_Data".F3.Btt_Up_Selected OR "DB_Data".F3.Btt_Down_Selected OR "DB_Data".F5.Btt_Down_Selected OR "DB_Data".F5.Btt_Up_Selected OR "DB_Data".F6.Btt_Down_Selected OR "DB_Data".F6.Btt_Up_Selected OR "DB_Data".F7.Btt_Down_Selected OR "DB_Data".F7.Btt_Up_Selected OR "DB_Data".F8.Btt_Down_Selected OR "DB_Data".F8.Btt_Up_Selected OR "DB_Data".F9.Btt_Down_Selected OR "DB_Data".F9.Btt_Up_Selected OR "DB_Data".F4.Btt_Down_Selected OR "DB_Data".F4.Btt_Up_Selected OR "DB_Data".F10.Btt_Down_Selected OR "DB_Data".F10.Btt_Up_Selected OR "DB_Data".F12.Btt_Down_Selected OR "DB_Data".F12.Btt_Up_Selected OR "DB_Data".F13.Btt_Down_Selected OR "DB_Data".F13.Btt_Up_Selected OR "DB_Data".F14.Btt_Down_Selected OR "DB_Data".F14.Btt_Up_Selected OR "DB_Data".F15.Btt_Down_Selected OR "DB_Data".F15.Btt_Up_Selected OR "DB_Data".F16.Btt_Down_Selected OR "DB_Data".F16.Btt_Up_Selected OR "DB_Data".F17.Btt_Down_Selected OR "DB_Data".F17.Btt_Up_Selected OR "DB_Data".F18.Btt_Down_Selected OR "DB_Data".F18.Btt_Up_Selected OR "DB_Data".F19.Btt_Down_Selected OR "DB_Data".F19.Btt_Up_Selected OR "DB_Data".F11.Btt_Down_Selected OR "DB_Data".F11.Btt_Up_Selected);
END_REGION

REGION Network 21: Ưu tiên đi lên hoặc đi xuống
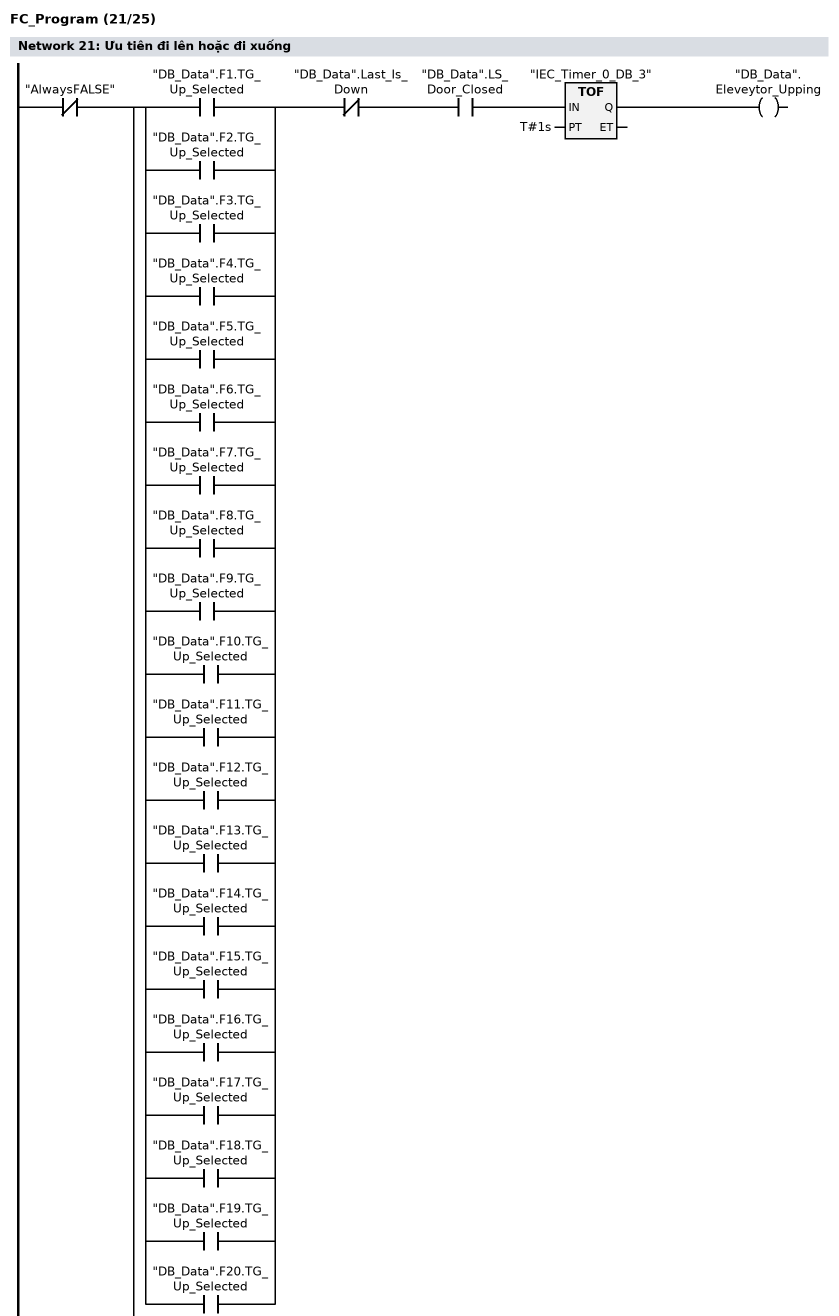
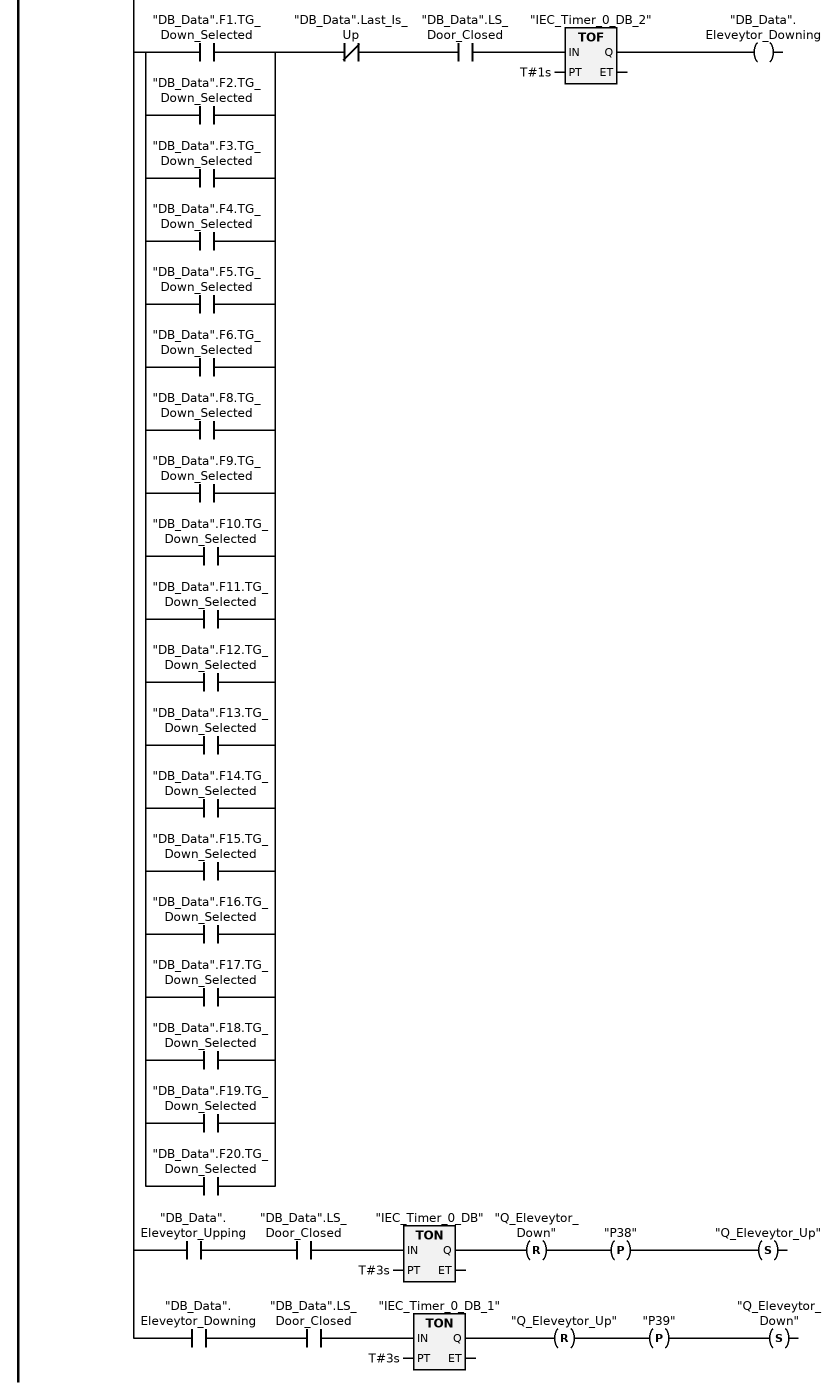
   "IEC_Timer_0_DB_3".TOF(IN := NOT "AlwaysFALSE" AND ("DB_Data".F1.TG_Up_Selected OR "DB_Data".F2.TG_Up_Selected OR "DB_Data".F3.TG_Up_Selected OR "DB_Data".F4.TG_Up_Selected OR "DB_Data".F5.TG_Up_Selected OR "DB_Data".F6.TG_Up_Selected OR "DB_Data".F7.TG_Up_Selected OR "DB_Data".F8.TG_Up_Selected OR "DB_Data".F9.TG_Up_Selected OR "DB_Data".F10.TG_Up_Selected OR "DB_Data".F11.TG_Up_Selected OR "DB_Data".F12.TG_Up_Selected OR "DB_Data".F13.TG_Up_Selected OR "DB_Data".F14.TG_Up_Selected OR "DB_Data".F15.TG_Up_Selected OR "DB_Data".F16.TG_Up_Selected OR "DB_Data".F17.TG_Up_Selected OR "DB_Data".F18.TG_Up_Selected OR "DB_Data".F19.TG_Up_Selected OR "DB_Data".F20.TG_Up_Selected) AND NOT "DB_Data".Last_Is_Down AND "DB_Data".LS_Door_Closed,
                          PT := T#1s);
   "DB_Data".Eleveytor_Upping := "IEC_Timer_0_DB_3".Q;
   "IEC_Timer_0_DB_2".TOF(IN := NOT "AlwaysFALSE" AND ("DB_Data".F1.TG_Down_Selected OR "DB_Data".F2.TG_Down_Selected OR "DB_Data".F3.TG_Down_Selected OR "DB_Data".F4.TG_Down_Selected OR "DB_Data".F5.TG_Down_Selected OR "DB_Data".F6.TG_Down_Selected OR "DB_Data".F8.TG_Down_Selected OR "DB_Data".F9.TG_Down_Selected OR "DB_Data".F10.TG_Down_Selected OR "DB_Data".F11.TG_Down_Selected OR "DB_Data".F12.TG_Down_Selected OR "DB_Data".F13.TG_Down_Selected OR "DB_Data".F14.TG_Down_Selected OR "DB_Data".F15.TG_Down_Selected OR "DB_Data".F16.TG_Down_Selected OR "DB_Data".F17.TG_Down_Selected OR "DB_Data".F18.TG_Down_Selected OR "DB_Data".F19.TG_Down_Selected OR "DB_Data".F20.TG_Down_Selected) AND NOT "DB_Data".Last_Is_Up AND "DB_Data".LS_Door_Closed,
                          PT := T#1s);
   "DB_Data".Eleveytor_Downing := "IEC_Timer_0_DB_2".Q;
   "IEC_Timer_0_DB".TON(IN := NOT "AlwaysFALSE" AND "DB_Data".Eleveytor_Upping AND "DB_Data".LS_Door_Closed,
                        PT := T#3s);
   IF "IEC_Timer_0_DB".Q THEN "Q_Eleveytor_Down" := FALSE; END_IF;
   #_w1 := "IEC_Timer_0_DB".Q AND NOT "P38";   // rising edge
   "P38" := "IEC_Timer_0_DB".Q;
   IF #_w1 THEN "Q_Eleveytor_Up" := TRUE; END_IF;
   "IEC_Timer_0_DB_1".TON(IN := NOT "AlwaysFALSE" AND "DB_Data".Eleveytor_Downing AND "DB_Data".LS_Door_Closed,
                          PT := T#3s);
   IF "IEC_Timer_0_DB_1".Q THEN "Q_Eleveytor_Up" := FALSE; END_IF;
   #_w2 := "IEC_Timer_0_DB_1".Q AND NOT "P39";   // rising edge
   "P39" := "IEC_Timer_0_DB_1".Q;
   IF #_w2 THEN "Q_Eleveytor_Down" := TRUE; END_IF;
END_REGION

REGION Network 22: Bit báo trạng thái trước đó
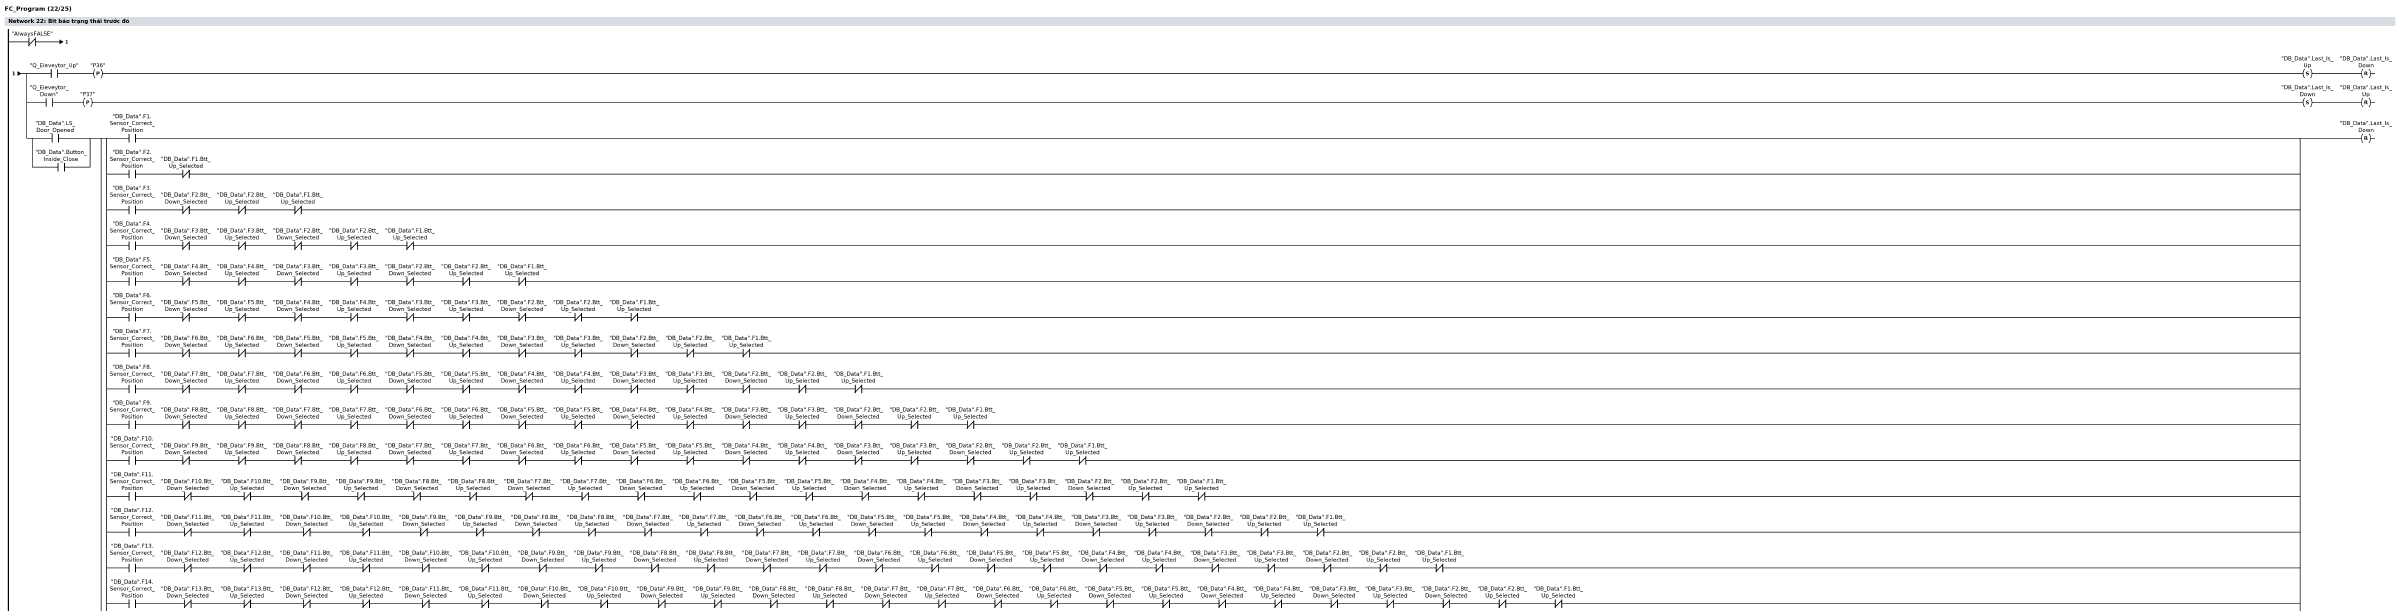
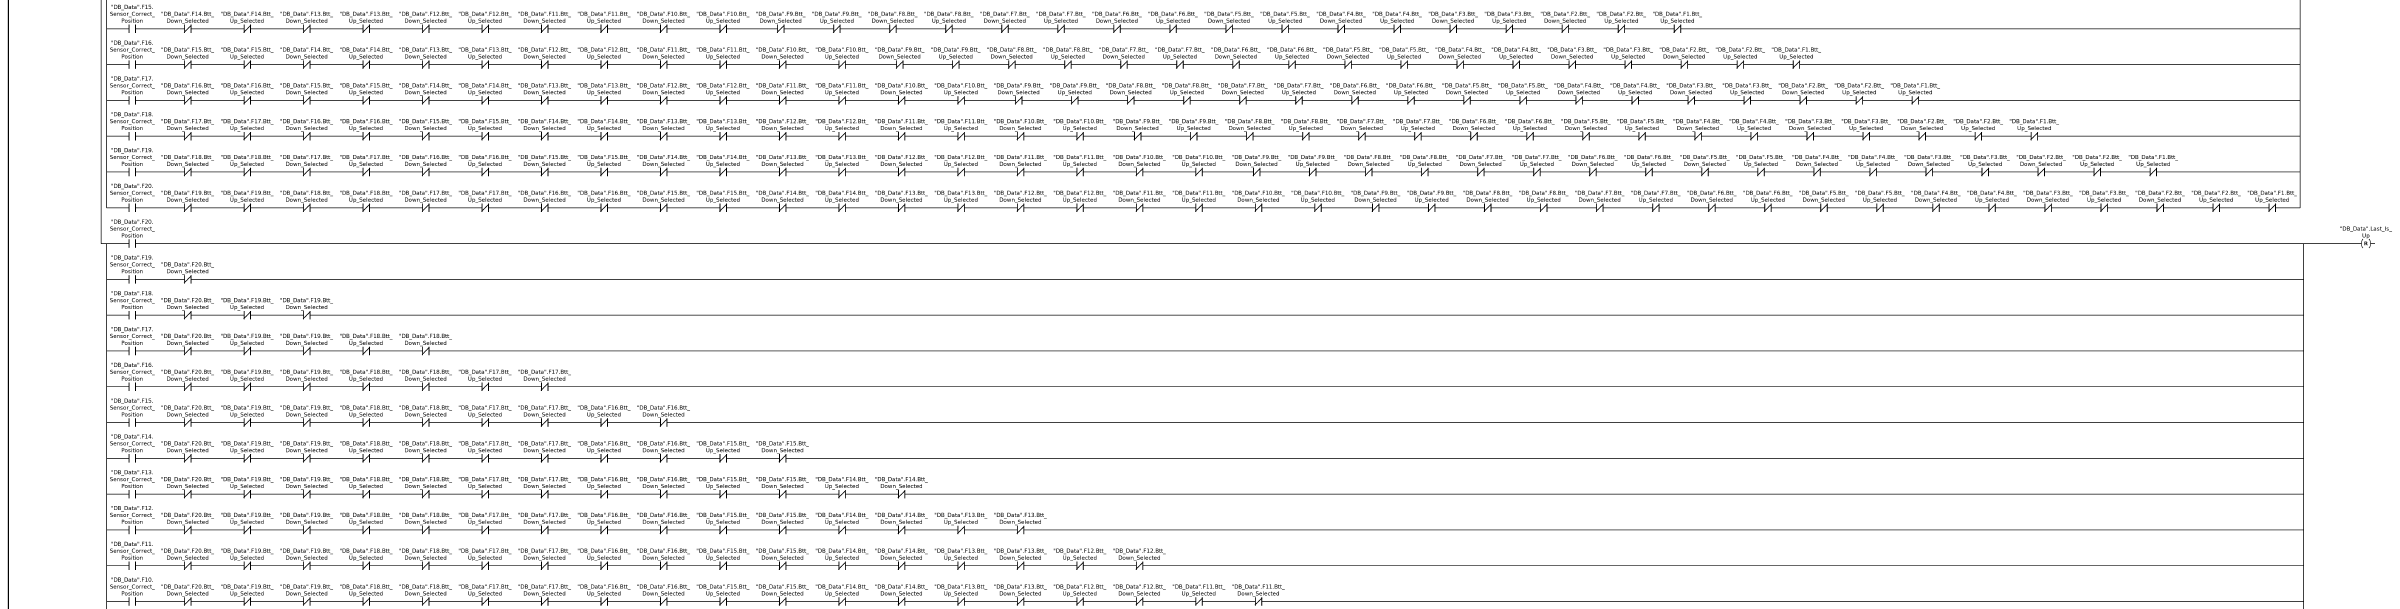
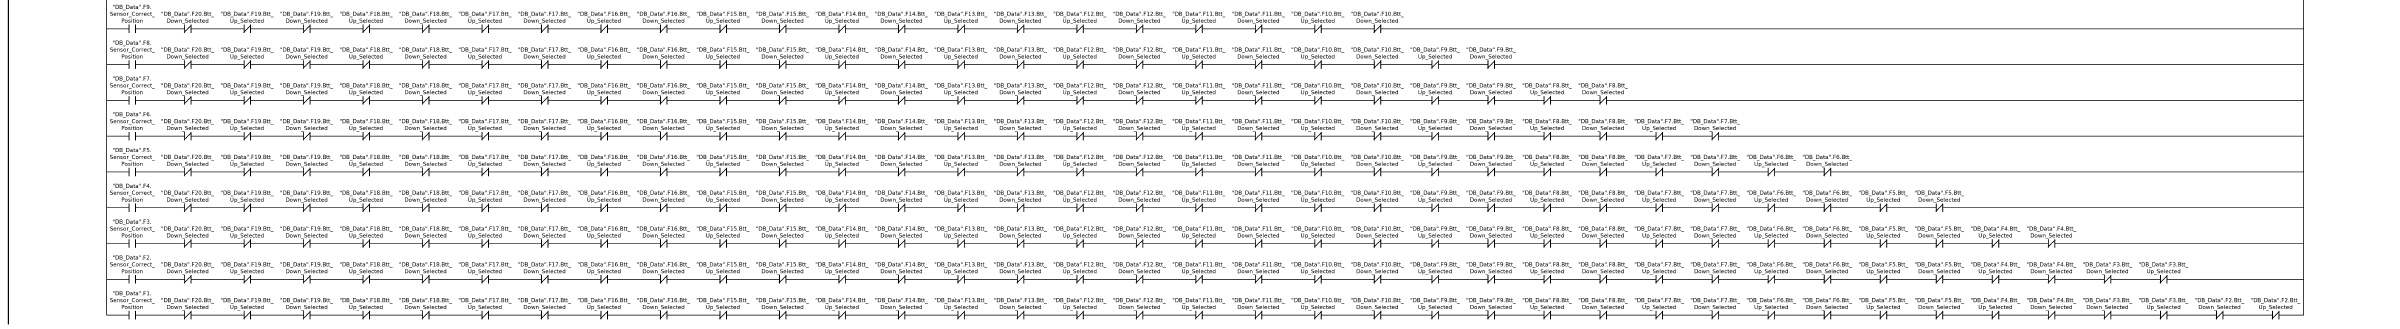
   RUNG wire#powerrail
      I_Contact( "AlwaysFALSE" )
      wire#w1
      Contact( "Q_Eleveytor_Up" )
      P_Trig( "P36" )
      S_Coil( "DB_Data".Last_Is_Up )
      R_Coil( "DB_Data".Last_Is_Down )
   END_RUNG
   RUNG wire#w1
      Contact( "Q_Eleveytor_Down" )
      P_Trig( "P37" )
      S_Coil( "DB_Data".Last_Is_Down )
      R_Coil( "DB_Data".Last_Is_Up )
   END_RUNG
   RUNG wire#w1
      Contact( "DB_Data".LS_Door_Opened )
      wire#w2
      Contact( "DB_Data".F1.Sensor_Correct_Position )
      wire#w3
      R_Coil( "DB_Data".Last_Is_Down )
   END_RUNG
   RUNG wire#w1
      Contact( "DB_Data".Button_Inside_Close )
   END_RUNG wire#w2
   RUNG wire#w2
      Contact( "DB_Data".F2.Sensor_Correct_Position )
      I_Contact( "DB_Data".F1.Btt_Up_Selected )
   END_RUNG wire#w3
   RUNG wire#w2
      Contact( "DB_Data".F3.Sensor_Correct_Position )
      I_Contact( "DB_Data".F2.Btt_Down_Selected )
      I_Contact( "DB_Data".F2.Btt_Up_Selected )
      I_Contact( "DB_Data".F1.Btt_Up_Selected )
   END_RUNG wire#w3
   RUNG wire#w2
      Contact( "DB_Data".F4.Sensor_Correct_Position )
      I_Contact( "DB_Data".F3.Btt_Down_Selected )
      I_Contact( "DB_Data".F3.Btt_Up_Selected )
      I_Contact( "DB_Data".F2.Btt_Down_Selected )
      I_Contact( "DB_Data".F2.Btt_Up_Selected )
      I_Contact( "DB_Data".F1.Btt_Up_Selected )
   END_RUNG wire#w3
   RUNG wire#w2
      Contact( "DB_Data".F5.Sensor_Correct_Position )
      I_Contact( "DB_Data".F4.Btt_Down_Selected )
      I_Contact( "DB_Data".F4.Btt_Up_Selected )
      I_Contact( "DB_Data".F3.Btt_Down_Selected )
      I_Contact( "DB_Data".F3.Btt_Up_Selected )
      I_Contact( "DB_Data".F2.Btt_Down_Selected )
      I_Contact( "DB_Data".F2.Btt_Up_Selected )
      I_Contact( "DB_Data".F1.Btt_Up_Selected )
   END_RUNG wire#w3
   RUNG wire#w2
      Contact( "DB_Data".F6.Sensor_Correct_Position )
      I_Contact( "DB_Data".F5.Btt_Down_Selected )
      I_Contact( "DB_Data".F5.Btt_Up_Selected )
      I_Contact( "DB_Data".F4.Btt_Down_Selected )
      I_Contact( "DB_Data".F4.Btt_Up_Selected )
      I_Contact( "DB_Data".F3.Btt_Down_Selected )
      I_Contact( "DB_Data".F3.Btt_Up_Selected )
      I_Contact( "DB_Data".F2.Btt_Down_Selected )
      I_Contact( "DB_Data".F2.Btt_Up_Selected )
      I_Contact( "DB_Data".F1.Btt_Up_Selected )
   END_RUNG wire#w3
   RUNG wire#w2
      Contact( "DB_Data".F7.Sensor_Correct_Position )
      I_Contact( "DB_Data".F6.Btt_Down_Selected )
      I_Contact( "DB_Data".F6.Btt_Up_Selected )
      I_Contact( "DB_Data".F5.Btt_Down_Selected )
      I_Contact( "DB_Data".F5.Btt_Up_Selected )
      I_Contact( "DB_Data".F4.Btt_Down_Selected )
      I_Contact( "DB_Data".F4.Btt_Up_Selected )
      I_Contact( "DB_Data".F3.Btt_Down_Selected )
      I_Contact( "DB_Data".F3.Btt_Up_Selected )
      I_Contact( "DB_Data".F2.Btt_Down_Selected )
      I_Contact( "DB_Data".F2.Btt_Up_Selected )
      I_Contact( "DB_Data".F1.Btt_Up_Selected )
   END_RUNG wire#w3
   RUNG wire#w2
      Contact( "DB_Data".F8.Sensor_Correct_Position )
      I_Contact( "DB_Data".F7.Btt_Down_Selected )
      I_Contact( "DB_Data".F7.Btt_Up_Selected )
      I_Contact( "DB_Data".F6.Btt_Down_Selected )
      I_Contact( "DB_Data".F6.Btt_Up_Selected )
      I_Contact( "DB_Data".F5.Btt_Down_Selected )
      I_Contact( "DB_Data".F5.Btt_Up_Selected )
      I_Contact( "DB_Data".F4.Btt_Down_Selected )
      I_Contact( "DB_Data".F4.Btt_Up_Selected )
      I_Contact( "DB_Data".F3.Btt_Down_Selected )
      I_Contact( "DB_Data".F3.Btt_Up_Selected )
      I_Contact( "DB_Data".F2.Btt_Down_Selected )
      I_Contact( "DB_Data".F2.Btt_Up_Selected )
      I_Contact( "DB_Data".F1.Btt_Up_Selected )
   END_RUNG wire#w3
   RUNG wire#w2
      Contact( "DB_Data".F9.Sensor_Correct_Position )
      I_Contact( "DB_Data".F8.Btt_Down_Selected )
      I_Contact( "DB_Data".F8.Btt_Up_Selected )
      I_Contact( "DB_Data".F7.Btt_Down_Selected )
      I_Contact( "DB_Data".F7.Btt_Up_Selected )
      I_Contact( "DB_Data".F6.Btt_Down_Selected )
      I_Contact( "DB_Data".F6.Btt_Up_Selected )
      I_Contact( "DB_Data".F5.Btt_Down_Selected )
      I_Contact( "DB_Data".F5.Btt_Up_Selected )
      I_Contact( "DB_Data".F4.Btt_Down_Selected )
      I_Contact( "DB_Data".F4.Btt_Up_Selected )
      I_Contact( "DB_Data".F3.Btt_Down_Selected )
      I_Contact( "DB_Data".F3.Btt_Up_Selected )
      I_Contact( "DB_Data".F2.Btt_Down_Selected )
      I_Contact( "DB_Data".F2.Btt_Up_Selected )
      I_Contact( "DB_Data".F1.Btt_Up_Selected )
   END_RUNG wire#w3
   RUNG wire#w2
      Contact( "DB_Data".F10.Sensor_Correct_Position )
      I_Contact( "DB_Data".F9.Btt_Down_Selected )
      I_Contact( "DB_Data".F9.Btt_Up_Selected )
      I_Contact( "DB_Data".F8.Btt_Down_Selected )
      I_Contact( "DB_Data".F8.Btt_Up_Selected )
      I_Contact( "DB_Data".F7.Btt_Down_Selected )
      I_Contact( "DB_Data".F7.Btt_Up_Selected )
      I_Contact( "DB_Data".F6.Btt_Down_Selected )
      I_Contact( "DB_Data".F6.Btt_Up_Selected )
      I_Contact( "DB_Data".F5.Btt_Down_Selected )
      I_Contact( "DB_Data".F5.Btt_Up_Selected )
      I_Contact( "DB_Data".F4.Btt_Down_Selected )
      I_Contact( "DB_Data".F4.Btt_Up_Selected )
      I_Contact( "DB_Data".F3.Btt_Down_Selected )
      I_Contact( "DB_Data".F3.Btt_Up_Selected )
      I_Contact( "DB_Data".F2.Btt_Down_Selected )
      I_Contact( "DB_Data".F2.Btt_Up_Selected )
      I_Contact( "DB_Data".F1.Btt_Up_Selected )
   END_RUNG wire#w3
   RUNG wire#w2
      Contact( "DB_Data".F11.Sensor_Correct_Position )
      I_Contact( "DB_Data".F10.Btt_Down_Selected )
      I_Contact( "DB_Data".F10.Btt_Up_Selected )
      I_Contact( "DB_Data".F9.Btt_Down_Selected )
      I_Contact( "DB_Data".F9.Btt_Up_Selected )
      I_Contact( "DB_Data".F8.Btt_Down_Selected )
      I_Contact( "DB_Data".F8.Btt_Up_Selected )
      I_Contact( "DB_Data".F7.Btt_Down_Selected )
      I_Contact( "DB_Data".F7.Btt_Up_Selected )
      I_Contact( "DB_Data".F6.Btt_Down_Selected )
      I_Contact( "DB_Data".F6.Btt_Up_Selected )
      I_Contact( "DB_Data".F5.Btt_Down_Selected )
      I_Contact( "DB_Data".F5.Btt_Up_Selected )
      I_Contact( "DB_Data".F4.Btt_Down_Selected )
      I_Contact( "DB_Data".F4.Btt_Up_Selected )
      I_Contact( "DB_Data".F3.Btt_Down_Selected )
      I_Contact( "DB_Data".F3.Btt_Up_Selected )
      I_Contact( "DB_Data".F2.Btt_Down_Selected )
      I_Contact( "DB_Data".F2.Btt_Up_Selected )
      I_Contact( "DB_Data".F1.Btt_Up_Selected )
   END_RUNG wire#w3
   RUNG wire#w2
      Contact( "DB_Data".F12.Sensor_Correct_Position )
      I_Contact( "DB_Data".F11.Btt_Down_Selected )
      I_Contact( "DB_Data".F11.Btt_Up_Selected )
      I_Contact( "DB_Data".F10.Btt_Down_Selected )
      I_Contact( "DB_Data".F10.Btt_Up_Selected )
      I_Contact( "DB_Data".F9.Btt_Down_Selected )
      I_Contact( "DB_Data".F9.Btt_Up_Selected )
      I_Contact( "DB_Data".F8.Btt_Down_Selected )
      I_Contact( "DB_Data".F8.Btt_Up_Selected )
      I_Contact( "DB_Data".F7.Btt_Down_Selected )
      I_Contact( "DB_Data".F7.Btt_Up_Selected )
      I_Contact( "DB_Data".F6.Btt_Down_Selected )
      I_Contact( "DB_Data".F6.Btt_Up_Selected )
      I_Contact( "DB_Data".F5.Btt_Down_Selected )
      I_Contact( "DB_Data".F5.Btt_Up_Selected )
      I_Contact( "DB_Data".F4.Btt_Down_Selected )
      I_Contact( "DB_Data".F4.Btt_Up_Selected )
      I_Contact( "DB_Data".F3.Btt_Down_Selected )
      I_Contact( "DB_Data".F3.Btt_Up_Selected )
      I_Contact( "DB_Data".F2.Btt_Down_Selected )
      I_Contact( "DB_Data".F2.Btt_Up_Selected )
      I_Contact( "DB_Data".F1.Btt_Up_Selected )
   END_RUNG wire#w3
   RUNG wire#w2
      Contact( "DB_Data".F13.Sensor_Correct_Position )
      I_Contact( "DB_Data".F12.Btt_Down_Selected )
      I_Contact( "DB_Data".F12.Btt_Up_Selected )
      I_Contact( "DB_Data".F11.Btt_Down_Selected )
      I_Contact( "DB_Data".F11.Btt_Up_Selected )
      I_Contact( "DB_Data".F10.Btt_Down_Selected )
      I_Contact( "DB_Data".F10.Btt_Up_Selected )
      I_Contact( "DB_Data".F9.Btt_Down_Selected )
      I_Contact( "DB_Data".F9.Btt_Up_Selected )
      I_Contact( "DB_Data".F8.Btt_Down_Selected )
      I_Contact( "DB_Data".F8.Btt_Up_Selected )
      I_Contact( "DB_Data".F7.Btt_Down_Selected )
      I_Contact( "DB_Data".F7.Btt_Up_Selected )
      I_Contact( "DB_Data".F6.Btt_Down_Selected )
      I_Contact( "DB_Data".F6.Btt_Up_Selected )
      I_Contact( "DB_Data".F5.Btt_Down_Selected )
      I_Contact( "DB_Data".F5.Btt_Up_Selected )
      I_Contact( "DB_Data".F4.Btt_Down_Selected )
      I_Contact( "DB_Data".F4.Btt_Up_Selected )
      I_Contact( "DB_Data".F3.Btt_Down_Selected )
      I_Contact( "DB_Data".F3.Btt_Up_Selected )
      I_Contact( "DB_Data".F2.Btt_Down_Selected )
      I_Contact( "DB_Data".F2.Btt_Up_Selected )
      I_Contact( "DB_Data".F1.Btt_Up_Selected )
   END_RUNG wire#w3
   RUNG wire#w2
      Contact( "DB_Data".F14.Sensor_Correct_Position )
      I_Contact( "DB_Data".F13.Btt_Down_Selected )
      I_Contact( "DB_Data".F13.Btt_Up_Selected )
      I_Contact( "DB_Data".F12.Btt_Down_Selected )
      I_Contact( "DB_Data".F12.Btt_Up_Selected )
      I_Contact( "DB_Data".F11.Btt_Down_Selected )
      I_Contact( "DB_Data".F11.Btt_Up_Selected )
      I_Contact( "DB_Data".F10.Btt_Down_Selected )
      I_Contact( "DB_Data".F10.Btt_Up_Selected )
      I_Contact( "DB_Data".F9.Btt_Down_Selected )
      I_Contact( "DB_Data".F9.Btt_Up_Selected )
      I_Contact( "DB_Data".F8.Btt_Down_Selected )
      I_Contact( "DB_Data".F8.Btt_Up_Selected )
      I_Contact( "DB_Data".F7.Btt_Down_Selected )
      I_Contact( "DB_Data".F7.Btt_Up_Selected )
      I_Contact( "DB_Data".F6.Btt_Down_Selected )
      I_Contact( "DB_Data".F6.Btt_Up_Selected )
      I_Contact( "DB_Data".F5.Btt_Down_Selected )
      I_Contact( "DB_Data".F5.Btt_Up_Selected )
      I_Contact( "DB_Data".F4.Btt_Down_Selected )
      I_Contact( "DB_Data".F4.Btt_Up_Selected )
      I_Contact( "DB_Data".F3.Btt_Down_Selected )
      I_Contact( "DB_Data".F3.Btt_Up_Selected )
      I_Contact( "DB_Data".F2.Btt_Down_Selected )
      I_Contact( "DB_Data".F2.Btt_Up_Selected )
      I_Contact( "DB_Data".F1.Btt_Up_Selected )
   END_RUNG wire#w3
   RUNG wire#w2
      Contact( "DB_Data".F15.Sensor_Correct_Position )
      I_Contact( "DB_Data".F14.Btt_Down_Selected )
      I_Contact( "DB_Data".F14.Btt_Up_Selected )
      I_Contact( "DB_Data".F13.Btt_Down_Selected )
      I_Contact( "DB_Data".F13.Btt_Up_Selected )
      I_Contact( "DB_Data".F12.Btt_Down_Selected )
      I_Contact( "DB_Data".F12.Btt_Up_Selected )
      I_Contact( "DB_Data".F11.Btt_Down_Selected )
      I_Contact( "DB_Data".F11.Btt_Up_Selected )
      I_Contact( "DB_Data".F10.Btt_Down_Selected )
      I_Contact( "DB_Data".F10.Btt_Up_Selected )
      I_Contact( "DB_Data".F9.Btt_Down_Selected )
      I_Contact( "DB_Data".F9.Btt_Up_Selected )
      I_Contact( "DB_Data".F8.Btt_Down_Selected )
      I_Contact( "DB_Data".F8.Btt_Up_Selected )
      I_Contact( "DB_Data".F7.Btt_Down_Selected )
      I_Contact( "DB_Data".F7.Btt_Up_Selected )
      I_Contact( "DB_Data".F6.Btt_Down_Selected )
      I_Contact( "DB_Data".F6.Btt_Up_Selected )
      I_Contact( "DB_Data".F5.Btt_Down_Selected )
      I_Contact( "DB_Data".F5.Btt_Up_Selected )
      I_Contact( "DB_Data".F4.Btt_Down_Selected )
      I_Contact( "DB_Data".F4.Btt_Up_Selected )
      I_Contact( "DB_Data".F3.Btt_Down_Selected )
      I_Contact( "DB_Data".F3.Btt_Up_Selected )
      I_Contact( "DB_Data".F2.Btt_Down_Selected )
      I_Contact( "DB_Data".F2.Btt_Up_Selected )
      I_Contact( "DB_Data".F1.Btt_Up_Selected )
   END_RUNG wire#w3
   RUNG wire#w2
      Contact( "DB_Data".F16.Sensor_Correct_Position )
      I_Contact( "DB_Data".F15.Btt_Down_Selected )
      I_Contact( "DB_Data".F15.Btt_Up_Selected )
      I_Contact( "DB_Data".F14.Btt_Down_Selected )
      I_Contact( "DB_Data".F14.Btt_Up_Selected )
      I_Contact( "DB_Data".F13.Btt_Down_Selected )
      I_Contact( "DB_Data".F13.Btt_Up_Selected )
      I_Contact( "DB_Data".F12.Btt_Down_Selected )
      I_Contact( "DB_Data".F12.Btt_Up_Selected )
      I_Contact( "DB_Data".F11.Btt_Down_Selected )
      I_Contact( "DB_Data".F11.Btt_Up_Selected )
      I_Contact( "DB_Data".F10.Btt_Down_Selected )
      I_Contact( "DB_Data".F10.Btt_Up_Selected )
      I_Contact( "DB_Data".F9.Btt_Down_Selected )
      I_Contact( "DB_Data".F9.Btt_Up_Selected )
      I_Contact( "DB_Data".F8.Btt_Down_Selected )
      I_Contact( "DB_Data".F8.Btt_Up_Selected )
      I_Contact( "DB_Data".F7.Btt_Down_Selected )
      I_Contact( "DB_Data".F7.Btt_Up_Selected )
      I_Contact( "DB_Data".F6.Btt_Down_Selected )
      I_Contact( "DB_Data".F6.Btt_Up_Selected )
      I_Contact( "DB_Data".F5.Btt_Down_Selected )
      I_Contact( "DB_Data".F5.Btt_Up_Selected )
      I_Contact( "DB_Data".F4.Btt_Down_Selected )
      I_Contact( "DB_Data".F4.Btt_Up_Selected )
      I_Contact( "DB_Data".F3.Btt_Down_Selected )
      I_Contact( "DB_Data".F3.Btt_Up_Selected )
      I_Contact( "DB_Data".F2.Btt_Down_Selected )
      I_Contact( "DB_Data".F2.Btt_Up_Selected )
      I_Contact( "DB_Data".F1.Btt_Up_Selected )
   END_RUNG wire#w3
   RUNG wire#w2
      Contact( "DB_Data".F17.Sensor_Correct_Position )
      I_Contact( "DB_Data".F16.Btt_Down_Selected )
      I_Contact( "DB_Data".F16.Btt_Up_Selected )
      I_Contact( "DB_Data".F15.Btt_Down_Selected )
      I_Contact( "DB_Data".F15.Btt_Up_Selected )
      I_Contact( "DB_Data".F14.Btt_Down_Selected )
      I_Contact( "DB_Data".F14.Btt_Up_Selected )
      I_Contact( "DB_Data".F13.Btt_Down_Selected )
      I_Contact( "DB_Data".F13.Btt_Up_Selected )
      I_Contact( "DB_Data".F12.Btt_Down_Selected )
      I_Contact( "DB_Data".F12.Btt_Up_Selected )
      I_Contact( "DB_Data".F11.Btt_Down_Selected )
      I_Contact( "DB_Data".F11.Btt_Up_Selected )
      I_Contact( "DB_Data".F10.Btt_Down_Selected )
      I_Contact( "DB_Data".F10.Btt_Up_Selected )
      I_Contact( "DB_Data".F9.Btt_Down_Selected )
      I_Contact( "DB_Data".F9.Btt_Up_Selected )
      I_Contact( "DB_Data".F8.Btt_Down_Selected )
      I_Contact( "DB_Data".F8.Btt_Up_Selected )
      I_Contact( "DB_Data".F7.Btt_Down_Selected )
      I_Contact( "DB_Data".F7.Btt_Up_Selected )
      I_Contact( "DB_Data".F6.Btt_Down_Selected )
      I_Contact( "DB_Data".F6.Btt_Up_Selected )
      I_Contact( "DB_Data".F5.Btt_Down_Selected )
      I_Contact( "DB_Data".F5.Btt_Up_Selected )
      I_Contact( "DB_Data".F4.Btt_Down_Selected )
      I_Contact( "DB_Data".F4.Btt_Up_Selected )
      I_Contact( "DB_Data".F3.Btt_Down_Selected )
      I_Contact( "DB_Data".F3.Btt_Up_Selected )
      I_Contact( "DB_Data".F2.Btt_Down_Selected )
      I_Contact( "DB_Data".F2.Btt_Up_Selected )
      I_Contact( "DB_Data".F1.Btt_Up_Selected )
   END_RUNG wire#w3
   RUNG wire#w2
      Contact( "DB_Data".F18.Sensor_Correct_Position )
      I_Contact( "DB_Data".F17.Btt_Down_Selected )
      I_Contact( "DB_Data".F17.Btt_Up_Selected )
      I_Contact( "DB_Data".F16.Btt_Down_Selected )
      I_Contact( "DB_Data".F16.Btt_Up_Selected )
      I_Contact( "DB_Data".F15.Btt_Down_Selected )
      I_Contact( "DB_Data".F15.Btt_Up_Selected )
      I_Contact( "DB_Data".F14.Btt_Down_Selected )
      I_Contact( "DB_Data".F14.Btt_Up_Selected )
      I_Contact( "DB_Data".F13.Btt_Down_Selected )
      I_Contact( "DB_Data".F13.Btt_Up_Selected )
      I_Contact( "DB_Data".F12.Btt_Down_Selected )
      I_Contact( "DB_Data".F12.Btt_Up_Selected )
      I_Contact( "DB_Data".F11.Btt_Down_Selected )
      I_Contact( "DB_Data".F11.Btt_Up_Selected )
      I_Contact( "DB_Data".F10.Btt_Down_Selected )
      I_Contact( "DB_Data".F10.Btt_Up_Selected )
      I_Contact( "DB_Data".F9.Btt_Down_Selected )
      I_Contact( "DB_Data".F9.Btt_Up_Selected )
      I_Contact( "DB_Data".F8.Btt_Down_Selected )
      I_Contact( "DB_Data".F8.Btt_Up_Selected )
      I_Contact( "DB_Data".F7.Btt_Down_Selected )
      I_Contact( "DB_Data".F7.Btt_Up_Selected )
      I_Contact( "DB_Data".F6.Btt_Down_Selected )
      I_Contact( "DB_Data".F6.Btt_Up_Selected )
      I_Contact( "DB_Data".F5.Btt_Down_Selected )
      I_Contact( "DB_Data".F5.Btt_Up_Selected )
      I_Contact( "DB_Data".F4.Btt_Down_Selected )
      I_Contact( "DB_Data".F4.Btt_Up_Selected )
      I_Contact( "DB_Data".F3.Btt_Down_Selected )
      I_Contact( "DB_Data".F3.Btt_Up_Selected )
      I_Contact( "DB_Data".F2.Btt_Down_Selected )
      I_Contact( "DB_Data".F2.Btt_Up_Selected )
      I_Contact( "DB_Data".F1.Btt_Up_Selected )
   END_RUNG wire#w3
   RUNG wire#w2
      Contact( "DB_Data".F19.Sensor_Correct_Position )
      I_Contact( "DB_Data".F18.Btt_Down_Selected )
      I_Contact( "DB_Data".F18.Btt_Up_Selected )
      I_Contact( "DB_Data".F17.Btt_Down_Selected )
      I_Contact( "DB_Data".F17.Btt_Up_Selected )
      I_Contact( "DB_Data".F16.Btt_Down_Selected )
      I_Contact( "DB_Data".F16.Btt_Up_Selected )
      I_Contact( "DB_Data".F15.Btt_Down_Selected )
      I_Contact( "DB_Data".F15.Btt_Up_Selected )
      I_Contact( "DB_Data".F14.Btt_Down_Selected )
      I_Contact( "DB_Data".F14.Btt_Up_Selected )
      I_Contact( "DB_Data".F13.Btt_Down_Selected )
      I_Contact( "DB_Data".F13.Btt_Up_Selected )
      I_Contact( "DB_Data".F12.Btt_Down_Selected )
      I_Contact( "DB_Data".F12.Btt_Up_Selected )
      I_Contact( "DB_Data".F11.Btt_Down_Selected )
      I_Contact( "DB_Data".F11.Btt_Up_Selected )
      I_Contact( "DB_Data".F10.Btt_Down_Selected )
      I_Contact( "DB_Data".F10.Btt_Up_Selected )
      I_Contact( "DB_Data".F9.Btt_Down_Selected )
      I_Contact( "DB_Data".F9.Btt_Up_Selected )
      I_Contact( "DB_Data".F8.Btt_Down_Selected )
      I_Contact( "DB_Data".F8.Btt_Up_Selected )
      I_Contact( "DB_Data".F7.Btt_Down_Selected )
      I_Contact( "DB_Data".F7.Btt_Up_Selected )
      I_Contact( "DB_Data".F6.Btt_Down_Selected )
      I_Contact( "DB_Data".F6.Btt_Up_Selected )
      I_Contact( "DB_Data".F5.Btt_Down_Selected )
      I_Contact( "DB_Data".F5.Btt_Up_Selected )
      I_Contact( "DB_Data".F4.Btt_Down_Selected )
      I_Contact( "DB_Data".F4.Btt_Up_Selected )
      I_Contact( "DB_Data".F3.Btt_Down_Selected )
      I_Contact( "DB_Data".F3.Btt_Up_Selected )
      I_Contact( "DB_Data".F2.Btt_Down_Selected )
      I_Contact( "DB_Data".F2.Btt_Up_Selected )
      I_Contact( "DB_Data".F1.Btt_Up_Selected )
   END_RUNG wire#w3
   RUNG wire#w2
      Contact( "DB_Data".F20.Sensor_Correct_Position )
      I_Contact( "DB_Data".F19.Btt_Down_Selected )
      I_Contact( "DB_Data".F19.Btt_Up_Selected )
      I_Contact( "DB_Data".F18.Btt_Down_Selected )
      I_Contact( "DB_Data".F18.Btt_Up_Selected )
      I_Contact( "DB_Data".F17.Btt_Down_Selected )
      I_Contact( "DB_Data".F17.Btt_Up_Selected )
      I_Contact( "DB_Data".F16.Btt_Down_Selected )
      I_Contact( "DB_Data".F16.Btt_Up_Selected )
      I_Contact( "DB_Data".F15.Btt_Down_Selected )
      I_Contact( "DB_Data".F15.Btt_Up_Selected )
      I_Contact( "DB_Data".F14.Btt_Down_Selected )
      I_Contact( "DB_Data".F14.Btt_Up_Selected )
      I_Contact( "DB_Data".F13.Btt_Down_Selected )
      I_Contact( "DB_Data".F13.Btt_Up_Selected )
      I_Contact( "DB_Data".F12.Btt_Down_Selected )
      I_Contact( "DB_Data".F12.Btt_Up_Selected )
      I_Contact( "DB_Data".F11.Btt_Down_Selected )
      I_Contact( "DB_Data".F11.Btt_Up_Selected )
      I_Contact( "DB_Data".F10.Btt_Down_Selected )
      I_Contact( "DB_Data".F10.Btt_Up_Selected )
      I_Contact( "DB_Data".F9.Btt_Down_Selected )
      I_Contact( "DB_Data".F9.Btt_Up_Selected )
      I_Contact( "DB_Data".F8.Btt_Down_Selected )
      I_Contact( "DB_Data".F8.Btt_Up_Selected )
      I_Contact( "DB_Data".F7.Btt_Down_Selected )
      I_Contact( "DB_Data".F7.Btt_Up_Selected )
      I_Contact( "DB_Data".F6.Btt_Down_Selected )
      I_Contact( "DB_Data".F6.Btt_Up_Selected )
      I_Contact( "DB_Data".F5.Btt_Down_Selected )
      I_Contact( "DB_Data".F5.Btt_Up_Selected )
      I_Contact( "DB_Data".F4.Btt_Down_Selected )
      I_Contact( "DB_Data".F4.Btt_Up_Selected )
      I_Contact( "DB_Data".F3.Btt_Down_Selected )
      I_Contact( "DB_Data".F3.Btt_Up_Selected )
      I_Contact( "DB_Data".F2.Btt_Down_Selected )
      I_Contact( "DB_Data".F2.Btt_Up_Selected )
      I_Contact( "DB_Data".F1.Btt_Up_Selected )
   END_RUNG wire#w3
   RUNG wire#w2
      Contact( "DB_Data".F20.Sensor_Correct_Position )
      wire#w4
      R_Coil( "DB_Data".Last_Is_Up )
   END_RUNG
   RUNG wire#w2
      Contact( "DB_Data".F19.Sensor_Correct_Position )
      I_Contact( "DB_Data".F20.Btt_Down_Selected )
   END_RUNG wire#w4
   RUNG wire#w2
      Contact( "DB_Data".F18.Sensor_Correct_Position )
      I_Contact( "DB_Data".F20.Btt_Down_Selected )
      I_Contact( "DB_Data".F19.Btt_Up_Selected )
      I_Contact( "DB_Data".F19.Btt_Down_Selected )
   END_RUNG wire#w4
   RUNG wire#w2
      Contact( "DB_Data".F17.Sensor_Correct_Position )
      I_Contact( "DB_Data".F20.Btt_Down_Selected )
      I_Contact( "DB_Data".F19.Btt_Up_Selected )
      I_Contact( "DB_Data".F19.Btt_Down_Selected )
      I_Contact( "DB_Data".F18.Btt_Up_Selected )
      I_Contact( "DB_Data".F18.Btt_Down_Selected )
   END_RUNG wire#w4
   RUNG wire#w2
      Contact( "DB_Data".F16.Sensor_Correct_Position )
      I_Contact( "DB_Data".F20.Btt_Down_Selected )
      I_Contact( "DB_Data".F19.Btt_Up_Selected )
      I_Contact( "DB_Data".F19.Btt_Down_Selected )
      I_Contact( "DB_Data".F18.Btt_Up_Selected )
      I_Contact( "DB_Data".F18.Btt_Down_Selected )
      I_Contact( "DB_Data".F17.Btt_Up_Selected )
      I_Contact( "DB_Data".F17.Btt_Down_Selected )
   END_RUNG wire#w4
   RUNG wire#w2
      Contact( "DB_Data".F15.Sensor_Correct_Position )
      I_Contact( "DB_Data".F20.Btt_Down_Selected )
      I_Contact( "DB_Data".F19.Btt_Up_Selected )
      I_Contact( "DB_Data".F19.Btt_Down_Selected )
      I_Contact( "DB_Data".F18.Btt_Up_Selected )
      I_Contact( "DB_Data".F18.Btt_Down_Selected )
      I_Contact( "DB_Data".F17.Btt_Up_Selected )
      I_Contact( "DB_Data".F17.Btt_Down_Selected )
      I_Contact( "DB_Data".F16.Btt_Up_Selected )
      I_Contact( "DB_Data".F16.Btt_Down_Selected )
   END_RUNG wire#w4
   RUNG wire#w2
      Contact( "DB_Data".F14.Sensor_Correct_Position )
      I_Contact( "DB_Data".F20.Btt_Down_Selected )
      I_Contact( "DB_Data".F19.Btt_Up_Selected )
      I_Contact( "DB_Data".F19.Btt_Down_Selected )
      I_Contact( "DB_Data".F18.Btt_Up_Selected )
      I_Contact( "DB_Data".F18.Btt_Down_Selected )
      I_Contact( "DB_Data".F17.Btt_Up_Selected )
      I_Contact( "DB_Data".F17.Btt_Down_Selected )
      I_Contact( "DB_Data".F16.Btt_Up_Selected )
      I_Contact( "DB_Data".F16.Btt_Down_Selected )
      I_Contact( "DB_Data".F15.Btt_Up_Selected )
      I_Contact( "DB_Data".F15.Btt_Down_Selected )
   END_RUNG wire#w4
   RUNG wire#w2
      Contact( "DB_Data".F13.Sensor_Correct_Position )
      I_Contact( "DB_Data".F20.Btt_Down_Selected )
      I_Contact( "DB_Data".F19.Btt_Up_Selected )
      I_Contact( "DB_Data".F19.Btt_Down_Selected )
      I_Contact( "DB_Data".F18.Btt_Up_Selected )
      I_Contact( "DB_Data".F18.Btt_Down_Selected )
      I_Contact( "DB_Data".F17.Btt_Up_Selected )
      I_Contact( "DB_Data".F17.Btt_Down_Selected )
      I_Contact( "DB_Data".F16.Btt_Up_Selected )
      I_Contact( "DB_Data".F16.Btt_Down_Selected )
      I_Contact( "DB_Data".F15.Btt_Up_Selected )
      I_Contact( "DB_Data".F15.Btt_Down_Selected )
      I_Contact( "DB_Data".F14.Btt_Up_Selected )
      I_Contact( "DB_Data".F14.Btt_Down_Selected )
   END_RUNG wire#w4
   RUNG wire#w2
      Contact( "DB_Data".F12.Sensor_Correct_Position )
      I_Contact( "DB_Data".F20.Btt_Down_Selected )
      I_Contact( "DB_Data".F19.Btt_Up_Selected )
      I_Contact( "DB_Data".F19.Btt_Down_Selected )
      I_Contact( "DB_Data".F18.Btt_Up_Selected )
      I_Contact( "DB_Data".F18.Btt_Down_Selected )
      I_Contact( "DB_Data".F17.Btt_Up_Selected )
      I_Contact( "DB_Data".F17.Btt_Down_Selected )
      I_Contact( "DB_Data".F16.Btt_Up_Selected )
      I_Contact( "DB_Data".F16.Btt_Down_Selected )
      I_Contact( "DB_Data".F15.Btt_Up_Selected )
      I_Contact( "DB_Data".F15.Btt_Down_Selected )
      I_Contact( "DB_Data".F14.Btt_Up_Selected )
      I_Contact( "DB_Data".F14.Btt_Down_Selected )
      I_Contact( "DB_Data".F13.Btt_Up_Selected )
      I_Contact( "DB_Data".F13.Btt_Down_Selected )
   END_RUNG wire#w4
   RUNG wire#w2
      Contact( "DB_Data".F11.Sensor_Correct_Position )
      I_Contact( "DB_Data".F20.Btt_Down_Selected )
      I_Contact( "DB_Data".F19.Btt_Up_Selected )
      I_Contact( "DB_Data".F19.Btt_Down_Selected )
      I_Contact( "DB_Data".F18.Btt_Up_Selected )
      I_Contact( "DB_Data".F18.Btt_Down_Selected )
      I_Contact( "DB_Data".F17.Btt_Up_Selected )
      I_Contact( "DB_Data".F17.Btt_Down_Selected )
      I_Contact( "DB_Data".F16.Btt_Up_Selected )
      I_Contact( "DB_Data".F16.Btt_Down_Selected )
      I_Contact( "DB_Data".F15.Btt_Up_Selected )
      I_Contact( "DB_Data".F15.Btt_Down_Selected )
      I_Contact( "DB_Data".F14.Btt_Up_Selected )
      I_Contact( "DB_Data".F14.Btt_Down_Selected )
      I_Contact( "DB_Data".F13.Btt_Up_Selected )
      I_Contact( "DB_Data".F13.Btt_Down_Selected )
      I_Contact( "DB_Data".F12.Btt_Up_Selected )
      I_Contact( "DB_Data".F12.Btt_Down_Selected )
   END_RUNG wire#w4
   RUNG wire#w2
      Contact( "DB_Data".F10.Sensor_Correct_Position )
      I_Contact( "DB_Data".F20.Btt_Down_Selected )
      I_Contact( "DB_Data".F19.Btt_Up_Selected )
      I_Contact( "DB_Data".F19.Btt_Down_Selected )
      I_Contact( "DB_Data".F18.Btt_Up_Selected )
      I_Contact( "DB_Data".F18.Btt_Down_Selected )
      I_Contact( "DB_Data".F17.Btt_Up_Selected )
      I_Contact( "DB_Data".F17.Btt_Down_Selected )
      I_Contact( "DB_Data".F16.Btt_Up_Selected )
      I_Contact( "DB_Data".F16.Btt_Down_Selected )
      I_Contact( "DB_Data".F15.Btt_Up_Selected )
      I_Contact( "DB_Data".F15.Btt_Down_Selected )
      I_Contact( "DB_Data".F14.Btt_Up_Selected )
      I_Contact( "DB_Data".F14.Btt_Down_Selected )
      I_Contact( "DB_Data".F13.Btt_Up_Selected )
      I_Contact( "DB_Data".F13.Btt_Down_Selected )
      I_Contact( "DB_Data".F12.Btt_Up_Selected )
      I_Contact( "DB_Data".F12.Btt_Down_Selected )
      I_Contact( "DB_Data".F11.Btt_Up_Selected )
      I_Contact( "DB_Data".F11.Btt_Down_Selected )
   END_RUNG wire#w4
   RUNG wire#w2
      Contact( "DB_Data".F9.Sensor_Correct_Position )
      I_Contact( "DB_Data".F20.Btt_Down_Selected )
      I_Contact( "DB_Data".F19.Btt_Up_Selected )
      I_Contact( "DB_Data".F19.Btt_Down_Selected )
      I_Contact( "DB_Data".F18.Btt_Up_Selected )
      I_Contact( "DB_Data".F18.Btt_Down_Selected )
      I_Contact( "DB_Data".F17.Btt_Up_Selected )
      I_Contact( "DB_Data".F17.Btt_Down_Selected )
      I_Contact( "DB_Data".F16.Btt_Up_Selected )
      I_Contact( "DB_Data".F16.Btt_Down_Selected )
      I_Contact( "DB_Data".F15.Btt_Up_Selected )
      I_Contact( "DB_Data".F15.Btt_Down_Selected )
      I_Contact( "DB_Data".F14.Btt_Up_Selected )
      I_Contact( "DB_Data".F14.Btt_Down_Selected )
      I_Contact( "DB_Data".F13.Btt_Up_Selected )
      I_Contact( "DB_Data".F13.Btt_Down_Selected )
      I_Contact( "DB_Data".F12.Btt_Up_Selected )
      I_Contact( "DB_Data".F12.Btt_Down_Selected )
      I_Contact( "DB_Data".F11.Btt_Up_Selected )
      I_Contact( "DB_Data".F11.Btt_Down_Selected )
      I_Contact( "DB_Data".F10.Btt_Up_Selected )
      I_Contact( "DB_Data".F10.Btt_Down_Selected )
   END_RUNG wire#w4
   RUNG wire#w2
      Contact( "DB_Data".F8.Sensor_Correct_Position )
      I_Contact( "DB_Data".F20.Btt_Down_Selected )
      I_Contact( "DB_Data".F19.Btt_Up_Selected )
      I_Contact( "DB_Data".F19.Btt_Down_Selected )
      I_Contact( "DB_Data".F18.Btt_Up_Selected )
      I_Contact( "DB_Data".F18.Btt_Down_Selected )
      I_Contact( "DB_Data".F17.Btt_Up_Selected )
      I_Contact( "DB_Data".F17.Btt_Down_Selected )
      I_Contact( "DB_Data".F16.Btt_Up_Selected )
      I_Contact( "DB_Data".F16.Btt_Down_Selected )
      I_Contact( "DB_Data".F15.Btt_Up_Selected )
      I_Contact( "DB_Data".F15.Btt_Down_Selected )
      I_Contact( "DB_Data".F14.Btt_Up_Selected )
      I_Contact( "DB_Data".F14.Btt_Down_Selected )
      I_Contact( "DB_Data".F13.Btt_Up_Selected )
      I_Contact( "DB_Data".F13.Btt_Down_Selected )
      I_Contact( "DB_Data".F12.Btt_Up_Selected )
      I_Contact( "DB_Data".F12.Btt_Down_Selected )
      I_Contact( "DB_Data".F11.Btt_Up_Selected )
      I_Contact( "DB_Data".F11.Btt_Down_Selected )
      I_Contact( "DB_Data".F10.Btt_Up_Selected )
      I_Contact( "DB_Data".F10.Btt_Down_Selected )
      I_Contact( "DB_Data".F9.Btt_Up_Selected )
      I_Contact( "DB_Data".F9.Btt_Down_Selected )
   END_RUNG wire#w4
   RUNG wire#w2
      Contact( "DB_Data".F7.Sensor_Correct_Position )
      I_Contact( "DB_Data".F20.Btt_Down_Selected )
      I_Contact( "DB_Data".F19.Btt_Up_Selected )
      I_Contact( "DB_Data".F19.Btt_Down_Selected )
      I_Contact( "DB_Data".F18.Btt_Up_Selected )
      I_Contact( "DB_Data".F18.Btt_Down_Selected )
      I_Contact( "DB_Data".F17.Btt_Up_Selected )
      I_Contact( "DB_Data".F17.Btt_Down_Selected )
      I_Contact( "DB_Data".F16.Btt_Up_Selected )
      I_Contact( "DB_Data".F16.Btt_Down_Selected )
      I_Contact( "DB_Data".F15.Btt_Up_Selected )
      I_Contact( "DB_Data".F15.Btt_Down_Selected )
      I_Contact( "DB_Data".F14.Btt_Up_Selected )
      I_Contact( "DB_Data".F14.Btt_Down_Selected )
      I_Contact( "DB_Data".F13.Btt_Up_Selected )
      I_Contact( "DB_Data".F13.Btt_Down_Selected )
      I_Contact( "DB_Data".F12.Btt_Up_Selected )
      I_Contact( "DB_Data".F12.Btt_Down_Selected )
      I_Contact( "DB_Data".F11.Btt_Up_Selected )
      I_Contact( "DB_Data".F11.Btt_Down_Selected )
      I_Contact( "DB_Data".F10.Btt_Up_Selected )
      I_Contact( "DB_Data".F10.Btt_Down_Selected )
      I_Contact( "DB_Data".F9.Btt_Up_Selected )
      I_Contact( "DB_Data".F9.Btt_Down_Selected )
      I_Contact( "DB_Data".F8.Btt_Up_Selected )
      I_Contact( "DB_Data".F8.Btt_Down_Selected )
   END_RUNG wire#w4
   RUNG wire#w2
      Contact( "DB_Data".F6.Sensor_Correct_Position )
      I_Contact( "DB_Data".F20.Btt_Down_Selected )
      I_Contact( "DB_Data".F19.Btt_Up_Selected )
      I_Contact( "DB_Data".F19.Btt_Down_Selected )
      I_Contact( "DB_Data".F18.Btt_Up_Selected )
      I_Contact( "DB_Data".F18.Btt_Down_Selected )
      I_Contact( "DB_Data".F17.Btt_Up_Selected )
      I_Contact( "DB_Data".F17.Btt_Down_Selected )
      I_Contact( "DB_Data".F16.Btt_Up_Selected )
      I_Contact( "DB_Data".F16.Btt_Down_Selected )
      I_Contact( "DB_Data".F15.Btt_Up_Selected )
      I_Contact( "DB_Data".F15.Btt_Down_Selected )
      I_Contact( "DB_Data".F14.Btt_Up_Selected )
      I_Contact( "DB_Data".F14.Btt_Down_Selected )
      I_Contact( "DB_Data".F13.Btt_Up_Selected )
      I_Contact( "DB_Data".F13.Btt_Down_Selected )
      I_Contact( "DB_Data".F12.Btt_Up_Selected )
      I_Contact( "DB_Data".F12.Btt_Down_Selected )
      I_Contact( "DB_Data".F11.Btt_Up_Selected )
      I_Contact( "DB_Data".F11.Btt_Down_Selected )
      I_Contact( "DB_Data".F10.Btt_Up_Selected )
      I_Contact( "DB_Data".F10.Btt_Down_Selected )
      I_Contact( "DB_Data".F9.Btt_Up_Selected )
      I_Contact( "DB_Data".F9.Btt_Down_Selected )
      I_Contact( "DB_Data".F8.Btt_Up_Selected )
      I_Contact( "DB_Data".F8.Btt_Down_Selected )
      I_Contact( "DB_Data".F7.Btt_Up_Selected )
      I_Contact( "DB_Data".F7.Btt_Down_Selected )
   END_RUNG wire#w4
   RUNG wire#w2
      Contact( "DB_Data".F5.Sensor_Correct_Position )
      I_Contact( "DB_Data".F20.Btt_Down_Selected )
      I_Contact( "DB_Data".F19.Btt_Up_Selected )
      I_Contact( "DB_Data".F19.Btt_Down_Selected )
      I_Contact( "DB_Data".F18.Btt_Up_Selected )
      I_Contact( "DB_Data".F18.Btt_Down_Selected )
      I_Contact( "DB_Data".F17.Btt_Up_Selected )
      I_Contact( "DB_Data".F17.Btt_Down_Selected )
      I_Contact( "DB_Data".F16.Btt_Up_Selected )
      I_Contact( "DB_Data".F16.Btt_Down_Selected )
      I_Contact( "DB_Data".F15.Btt_Up_Selected )
      I_Contact( "DB_Data".F15.Btt_Down_Selected )
      I_Contact( "DB_Data".F14.Btt_Up_Selected )
      I_Contact( "DB_Data".F14.Btt_Down_Selected )
      I_Contact( "DB_Data".F13.Btt_Up_Selected )
      I_Contact( "DB_Data".F13.Btt_Down_Selected )
      I_Contact( "DB_Data".F12.Btt_Up_Selected )
      I_Contact( "DB_Data".F12.Btt_Down_Selected )
      I_Contact( "DB_Data".F11.Btt_Up_Selected )
      I_Contact( "DB_Data".F11.Btt_Down_Selected )
      I_Contact( "DB_Data".F10.Btt_Up_Selected )
      I_Contact( "DB_Data".F10.Btt_Down_Selected )
      I_Contact( "DB_Data".F9.Btt_Up_Selected )
      I_Contact( "DB_Data".F9.Btt_Down_Selected )
      I_Contact( "DB_Data".F8.Btt_Up_Selected )
      I_Contact( "DB_Data".F8.Btt_Down_Selected )
      I_Contact( "DB_Data".F7.Btt_Up_Selected )
      I_Contact( "DB_Data".F7.Btt_Down_Selected )
      I_Contact( "DB_Data".F6.Btt_Up_Selected )
      I_Contact( "DB_Data".F6.Btt_Down_Selected )
   END_RUNG wire#w4
   RUNG wire#w2
      Contact( "DB_Data".F4.Sensor_Correct_Position )
      I_Contact( "DB_Data".F20.Btt_Down_Selected )
      I_Contact( "DB_Data".F19.Btt_Up_Selected )
      I_Contact( "DB_Data".F19.Btt_Down_Selected )
      I_Contact( "DB_Data".F18.Btt_Up_Selected )
      I_Contact( "DB_Data".F18.Btt_Down_Selected )
      I_Contact( "DB_Data".F17.Btt_Up_Selected )
      I_Contact( "DB_Data".F17.Btt_Down_Selected )
      I_Contact( "DB_Data".F16.Btt_Up_Selected )
      I_Contact( "DB_Data".F16.Btt_Down_Selected )
      I_Contact( "DB_Data".F15.Btt_Up_Selected )
      I_Contact( "DB_Data".F15.Btt_Down_Selected )
      I_Contact( "DB_Data".F14.Btt_Up_Selected )
      I_Contact( "DB_Data".F14.Btt_Down_Selected )
      I_Contact( "DB_Data".F13.Btt_Up_Selected )
      I_Contact( "DB_Data".F13.Btt_Down_Selected )
      I_Contact( "DB_Data".F12.Btt_Up_Selected )
      I_Contact( "DB_Data".F12.Btt_Down_Selected )
      I_Contact( "DB_Data".F11.Btt_Up_Selected )
      I_Contact( "DB_Data".F11.Btt_Down_Selected )
      I_Contact( "DB_Data".F10.Btt_Up_Selected )
      I_Contact( "DB_Data".F10.Btt_Down_Selected )
      I_Contact( "DB_Data".F9.Btt_Up_Selected )
      I_Contact( "DB_Data".F9.Btt_Down_Selected )
      I_Contact( "DB_Data".F8.Btt_Up_Selected )
      I_Contact( "DB_Data".F8.Btt_Down_Selected )
      I_Contact( "DB_Data".F7.Btt_Up_Selected )
      I_Contact( "DB_Data".F7.Btt_Down_Selected )
      I_Contact( "DB_Data".F6.Btt_Up_Selected )
      I_Contact( "DB_Data".F6.Btt_Down_Selected )
      I_Contact( "DB_Data".F5.Btt_Up_Selected )
      I_Contact( "DB_Data".F5.Btt_Down_Selected )
   END_RUNG wire#w4
   RUNG wire#w2
      Contact( "DB_Data".F3.Sensor_Correct_Position )
      I_Contact( "DB_Data".F20.Btt_Down_Selected )
      I_Contact( "DB_Data".F19.Btt_Up_Selected )
      I_Contact( "DB_Data".F19.Btt_Down_Selected )
      I_Contact( "DB_Data".F18.Btt_Up_Selected )
      I_Contact( "DB_Data".F18.Btt_Down_Selected )
      I_Contact( "DB_Data".F17.Btt_Up_Selected )
      I_Contact( "DB_Data".F17.Btt_Down_Selected )
      I_Contact( "DB_Data".F16.Btt_Up_Selected )
      I_Contact( "DB_Data".F16.Btt_Down_Selected )
      I_Contact( "DB_Data".F15.Btt_Up_Selected )
      I_Contact( "DB_Data".F15.Btt_Down_Selected )
      I_Contact( "DB_Data".F14.Btt_Up_Selected )
      I_Contact( "DB_Data".F14.Btt_Down_Selected )
      I_Contact( "DB_Data".F13.Btt_Up_Selected )
      I_Contact( "DB_Data".F13.Btt_Down_Selected )
      I_Contact( "DB_Data".F12.Btt_Up_Selected )
      I_Contact( "DB_Data".F12.Btt_Down_Selected )
      I_Contact( "DB_Data".F11.Btt_Up_Selected )
      I_Contact( "DB_Data".F11.Btt_Down_Selected )
      I_Contact( "DB_Data".F10.Btt_Up_Selected )
      I_Contact( "DB_Data".F10.Btt_Down_Selected )
      I_Contact( "DB_Data".F9.Btt_Up_Selected )
      I_Contact( "DB_Data".F9.Btt_Down_Selected )
      I_Contact( "DB_Data".F8.Btt_Up_Selected )
      I_Contact( "DB_Data".F8.Btt_Down_Selected )
      I_Contact( "DB_Data".F7.Btt_Up_Selected )
      I_Contact( "DB_Data".F7.Btt_Down_Selected )
      I_Contact( "DB_Data".F6.Btt_Up_Selected )
      I_Contact( "DB_Data".F6.Btt_Down_Selected )
      I_Contact( "DB_Data".F5.Btt_Up_Selected )
      I_Contact( "DB_Data".F5.Btt_Down_Selected )
      I_Contact( "DB_Data".F4.Btt_Up_Selected )
      I_Contact( "DB_Data".F4.Btt_Down_Selected )
   END_RUNG wire#w4
   RUNG wire#w2
      Contact( "DB_Data".F2.Sensor_Correct_Position )
      I_Contact( "DB_Data".F20.Btt_Down_Selected )
      I_Contact( "DB_Data".F19.Btt_Up_Selected )
      I_Contact( "DB_Data".F19.Btt_Down_Selected )
      I_Contact( "DB_Data".F18.Btt_Up_Selected )
      I_Contact( "DB_Data".F18.Btt_Down_Selected )
      I_Contact( "DB_Data".F17.Btt_Up_Selected )
      I_Contact( "DB_Data".F17.Btt_Down_Selected )
      I_Contact( "DB_Data".F16.Btt_Up_Selected )
      I_Contact( "DB_Data".F16.Btt_Down_Selected )
      I_Contact( "DB_Data".F15.Btt_Up_Selected )
      I_Contact( "DB_Data".F15.Btt_Down_Selected )
      I_Contact( "DB_Data".F14.Btt_Up_Selected )
      I_Contact( "DB_Data".F14.Btt_Down_Selected )
      I_Contact( "DB_Data".F13.Btt_Up_Selected )
      I_Contact( "DB_Data".F13.Btt_Down_Selected )
      I_Contact( "DB_Data".F12.Btt_Up_Selected )
      I_Contact( "DB_Data".F12.Btt_Down_Selected )
      I_Contact( "DB_Data".F11.Btt_Up_Selected )
      I_Contact( "DB_Data".F11.Btt_Down_Selected )
      I_Contact( "DB_Data".F10.Btt_Up_Selected )
      I_Contact( "DB_Data".F10.Btt_Down_Selected )
      I_Contact( "DB_Data".F9.Btt_Up_Selected )
      I_Contact( "DB_Data".F9.Btt_Down_Selected )
      I_Contact( "DB_Data".F8.Btt_Up_Selected )
      I_Contact( "DB_Data".F8.Btt_Down_Selected )
      I_Contact( "DB_Data".F7.Btt_Up_Selected )
      I_Contact( "DB_Data".F7.Btt_Down_Selected )
      I_Contact( "DB_Data".F6.Btt_Up_Selected )
      I_Contact( "DB_Data".F6.Btt_Down_Selected )
      I_Contact( "DB_Data".F5.Btt_Up_Selected )
      I_Contact( "DB_Data".F5.Btt_Down_Selected )
      I_Contact( "DB_Data".F4.Btt_Up_Selected )
      I_Contact( "DB_Data".F4.Btt_Down_Selected )
      I_Contact( "DB_Data".F3.Btt_Down_Selected )
      I_Contact( "DB_Data".F3.Btt_Up_Selected )
   END_RUNG wire#w4
   RUNG wire#w2
      Contact( "DB_Data".F1.Sensor_Correct_Position )
      I_Contact( "DB_Data".F20.Btt_Down_Selected )
      I_Contact( "DB_Data".F19.Btt_Up_Selected )
      I_Contact( "DB_Data".F19.Btt_Down_Selected )
      I_Contact( "DB_Data".F18.Btt_Up_Selected )
      I_Contact( "DB_Data".F18.Btt_Down_Selected )
      I_Contact( "DB_Data".F17.Btt_Up_Selected )
      I_Contact( "DB_Data".F17.Btt_Down_Selected )
      I_Contact( "DB_Data".F16.Btt_Up_Selected )
      I_Contact( "DB_Data".F16.Btt_Down_Selected )
      I_Contact( "DB_Data".F15.Btt_Up_Selected )
      I_Contact( "DB_Data".F15.Btt_Down_Selected )
      I_Contact( "DB_Data".F14.Btt_Up_Selected )
      I_Contact( "DB_Data".F14.Btt_Down_Selected )
      I_Contact( "DB_Data".F13.Btt_Up_Selected )
      I_Contact( "DB_Data".F13.Btt_Down_Selected )
      I_Contact( "DB_Data".F12.Btt_Up_Selected )
      I_Contact( "DB_Data".F12.Btt_Down_Selected )
      I_Contact( "DB_Data".F11.Btt_Up_Selected )
      I_Contact( "DB_Data".F11.Btt_Down_Selected )
      I_Contact( "DB_Data".F10.Btt_Up_Selected )
      I_Contact( "DB_Data".F10.Btt_Down_Selected )
      I_Contact( "DB_Data".F9.Btt_Up_Selected )
      I_Contact( "DB_Data".F9.Btt_Down_Selected )
      I_Contact( "DB_Data".F8.Btt_Up_Selected )
      I_Contact( "DB_Data".F8.Btt_Down_Selected )
      I_Contact( "DB_Data".F7.Btt_Up_Selected )
      I_Contact( "DB_Data".F7.Btt_Down_Selected )
      I_Contact( "DB_Data".F6.Btt_Up_Selected )
      I_Contact( "DB_Data".F6.Btt_Down_Selected )
      I_Contact( "DB_Data".F5.Btt_Up_Selected )
      I_Contact( "DB_Data".F5.Btt_Down_Selected )
      I_Contact( "DB_Data".F4.Btt_Up_Selected )
      I_Contact( "DB_Data".F4.Btt_Down_Selected )
      I_Contact( "DB_Data".F3.Btt_Down_Selected )
      I_Contact( "DB_Data".F3.Btt_Up_Selected )
      I_Contact( "DB_Data".F2.Btt_Down_Selected )
      I_Contact( "DB_Data".F2.Btt_Up_Selected )
   END_RUNG wire#w4
   // the same network as SCL:
   #_w1 := NOT "AlwaysFALSE" AND "Q_Eleveytor_Up";
   #_w2 := #_w1 AND NOT "P36";   // rising edge
   "P36" := #_w1;
   IF #_w2 THEN
       "DB_Data".Last_Is_Up := TRUE;
       "DB_Data".Last_Is_Down := FALSE;
   END_IF;
   #_w3 := NOT "AlwaysFALSE" AND "Q_Eleveytor_Down";
   #_w4 := #_w3 AND NOT "P37";   // rising edge
   "P37" := #_w3;
   IF #_w4 THEN
       "DB_Data".Last_Is_Down := TRUE;
       "DB_Data".Last_Is_Up := FALSE;
   END_IF;
   #_w5 := NOT "AlwaysFALSE" AND ("DB_Data".LS_Door_Opened OR "DB_Data".Button_Inside_Close);
   IF #_w5 AND ("DB_Data".F1.Sensor_Correct_Position OR ("DB_Data".F2.Sensor_Correct_Position AND NOT "DB_Data".F1.Btt_Up_Selected) OR ("DB_Data".F3.Sensor_Correct_Position AND NOT "DB_Data".F2.Btt_Down_Selected AND NOT "DB_Data".F2.Btt_Up_Selected AND NOT "DB_Data".F1.Btt_Up_Selected) OR ("DB_Data".F4.Sensor_Correct_Position AND NOT "DB_Data".F3.Btt_Down_Selected AND NOT "DB_Data".F3.Btt_Up_Selected AND NOT "DB_Data".F2.Btt_Down_Selected AND NOT "DB_Data".F2.Btt_Up_Selected AND NOT "DB_Data".F1.Btt_Up_Selected) OR ("DB_Data".F5.Sensor_Correct_Position AND NOT "DB_Data".F4.Btt_Down_Selected AND NOT "DB_Data".F4.Btt_Up_Selected AND NOT "DB_Data".F3.Btt_Down_Selected AND NOT "DB_Data".F3.Btt_Up_Selected AND NOT "DB_Data".F2.Btt_Down_Selected AND NOT "DB_Data".F2.Btt_Up_Selected AND NOT "DB_Data".F1.Btt_Up_Selected) OR ("DB_Data".F6.Sensor_Correct_Position AND NOT "DB_Data".F5.Btt_Down_Selected AND NOT "DB_Data".F5.Btt_Up_Selected AND NOT "DB_Data".F4.Btt_Down_Selected AND NOT "DB_Data".F4.Btt_Up_Selected AND NOT "DB_Data".F3.Btt_Down_Selected AND NOT "DB_Data".F3.Btt_Up_Selected AND NOT "DB_Data".F2.Btt_Down_Selected AND NOT "DB_Data".F2.Btt_Up_Selected AND NOT "DB_Data".F1.Btt_Up_Selected) OR ("DB_Data".F7.Sensor_Correct_Position AND NOT "DB_Data".F6.Btt_Down_Selected AND NOT "DB_Data".F6.Btt_Up_Selected AND NOT "DB_Data".F5.Btt_Down_Selected AND NOT "DB_Data".F5.Btt_Up_Selected AND NOT "DB_Data".F4.Btt_Down_Selected AND NOT "DB_Data".F4.Btt_Up_Selected AND NOT "DB_Data".F3.Btt_Down_Selected AND NOT "DB_Data".F3.Btt_Up_Selected AND NOT "DB_Data".F2.Btt_Down_Selected AND NOT "DB_Data".F2.Btt_Up_Selected AND NOT "DB_Data".F1.Btt_Up_Selected) OR ("DB_Data".F8.Sensor_Correct_Position AND NOT "DB_Data".F7.Btt_Down_Selected AND NOT "DB_Data".F7.Btt_Up_Selected AND NOT "DB_Data".F6.Btt_Down_Selected AND NOT "DB_Data".F6.Btt_Up_Selected AND NOT "DB_Data".F5.Btt_Down_Selected AND NOT "DB_Data".F5.Btt_Up_Selected AND NOT "DB_Data".F4.Btt_Down_Selected AND NOT "DB_Data".F4.Btt_Up_Selected AND NOT "DB_Data".F3.Btt_Down_Selected AND NOT "DB_Data".F3.Btt_Up_Selected AND NOT "DB_Data".F2.Btt_Down_Selected AND NOT "DB_Data".F2.Btt_Up_Selected AND NOT "DB_Data".F1.Btt_Up_Selected) OR ("DB_Data".F9.Sensor_Correct_Position AND NOT "DB_Data".F8.Btt_Down_Selected AND NOT "DB_Data".F8.Btt_Up_Selected AND NOT "DB_Data".F7.Btt_Down_Selected AND NOT "DB_Data".F7.Btt_Up_Selected AND NOT "DB_Data".F6.Btt_Down_Selected AND NOT "DB_Data".F6.Btt_Up_Selected AND NOT "DB_Data".F5.Btt_Down_Selected AND NOT "DB_Data".F5.Btt_Up_Selected AND NOT "DB_Data".F4.Btt_Down_Selected AND NOT "DB_Data".F4.Btt_Up_Selected AND NOT "DB_Data".F3.Btt_Down_Selected AND NOT "DB_Data".F3.Btt_Up_Selected AND NOT "DB_Data".F2.Btt_Down_Selected AND NOT "DB_Data".F2.Btt_Up_Selected AND NOT "DB_Data".F1.Btt_Up_Selected) OR ("DB_Data".F10.Sensor_Correct_Position AND NOT "DB_Data".F9.Btt_Down_Selected AND NOT "DB_Data".F9.Btt_Up_Selected AND NOT "DB_Data".F8.Btt_Down_Selected AND NOT "DB_Data".F8.Btt_Up_Selected AND NOT "DB_Data".F7.Btt_Down_Selected AND NOT "DB_Data".F7.Btt_Up_Selected AND NOT "DB_Data".F6.Btt_Down_Selected AND NOT "DB_Data".F6.Btt_Up_Selected AND NOT "DB_Data".F5.Btt_Down_Selected AND NOT "DB_Data".F5.Btt_Up_Selected AND NOT "DB_Data".F4.Btt_Down_Selected AND NOT "DB_Data".F4.Btt_Up_Selected AND NOT "DB_Data".F3.Btt_Down_Selected AND NOT "DB_Data".F3.Btt_Up_Selected AND NOT "DB_Data".F2.Btt_Down_Selected AND NOT "DB_Data".F2.Btt_Up_Selected AND NOT "DB_Data".F1.Btt_Up_Selected) OR ("DB_Data".F11.Sensor_Correct_Position AND NOT "DB_Data".F10.Btt_Down_Selected AND NOT "DB_Data".F10.Btt_Up_Selected AND NOT "DB_Data".F9.Btt_Down_Selected AND NOT "DB_Data".F9.Btt_Up_Selected AND NOT "DB_Data".F8.Btt_Down_Selected AND NOT "DB_Data".F8.Btt_Up_Selected AND NOT "DB_Data".F7.Btt_Down_Selected AND NOT "DB_Data".F7.Btt_Up_Selected AND NOT "DB_Data".F6.Btt_Down_Selected AND NOT "DB_Data".F6.Btt_Up_Selected AND NOT "DB_Data".F5.Btt_Down_Selected AND NOT "DB_Data".F5.Btt_Up_Selected AND NOT "DB_Data".F4.Btt_Down_Selected AND NOT "DB_Data".F4.Btt_Up_Selected AND NOT "DB_Data".F3.Btt_Down_Selected AND NOT "DB_Data".F3.Btt_Up_Selected AND NOT "DB_Data".F2.Btt_Down_Selected AND NOT "DB_Data".F2.Btt_Up_Selected AND NOT "DB_Data".F1.Btt_Up_Selected) OR ("DB_Data".F12.Sensor_Correct_Position AND NOT "DB_Data".F11.Btt_Down_Selected AND NOT "DB_Data".F11.Btt_Up_Selected AND NOT "DB_Data".F10.Btt_Down_Selected AND NOT "DB_Data".F10.Btt_Up_Selected AND NOT "DB_Data".F9.Btt_Down_Selected AND NOT "DB_Data".F9.Btt_Up_Selected AND NOT "DB_Data".F8.Btt_Down_Selected AND NOT "DB_Data".F8.Btt_Up_Selected AND NOT "DB_Data".F7.Btt_Down_Selected AND NOT "DB_Data".F7.Btt_Up_Selected AND NOT "DB_Data".F6.Btt_Down_Selected AND NOT "DB_Data".F6.Btt_Up_Selected AND NOT "DB_Data".F5.Btt_Down_Selected AND NOT "DB_Data".F5.Btt_Up_Selected AND NOT "DB_Data".F4.Btt_Down_Selected AND NOT "DB_Data".F4.Btt_Up_Selected AND NOT "DB_Data".F3.Btt_Down_Selected AND NOT "DB_Data".F3.Btt_Up_Selected AND NOT "DB_Data".F2.Btt_Down_Selected AND NOT "DB_Data".F2.Btt_Up_Selected AND NOT "DB_Data".F1.Btt_Up_Selected) OR ("DB_Data".F13.Sensor_Correct_Position AND NOT "DB_Data".F12.Btt_Down_Selected AND NOT "DB_Data".F12.Btt_Up_Selected AND NOT "DB_Data".F11.Btt_Down_Selected AND NOT "DB_Data".F11.Btt_Up_Selected AND NOT "DB_Data".F10.Btt_Down_Selected AND NOT "DB_Data".F10.Btt_Up_Selected AND NOT "DB_Data".F9.Btt_Down_Selected AND NOT "DB_Data".F9.Btt_Up_Selected AND NOT "DB_Data".F8.Btt_Down_Selected AND NOT "DB_Data".F8.Btt_Up_Selected AND NOT "DB_Data".F7.Btt_Down_Selected AND NOT "DB_Data".F7.Btt_Up_Selected AND NOT "DB_Data".F6.Btt_Down_Selected AND NOT "DB_Data".F6.Btt_Up_Selected AND NOT "DB_Data".F5.Btt_Down_Selected AND NOT "DB_Data".F5.Btt_Up_Selected AND NOT "DB_Data".F4.Btt_Down_Selected AND NOT "DB_Data".F4.Btt_Up_Selected AND NOT "DB_Data".F3.Btt_Down_Selected AND NOT "DB_Data".F3.Btt_Up_Selected AND NOT "DB_Data".F2.Btt_Down_Selected AND NOT "DB_Data".F2.Btt_Up_Selected AND NOT "DB_Data".F1.Btt_Up_Selected) OR ("DB_Data".F14.Sensor_Correct_Position AND NOT "DB_Data".F13.Btt_Down_Selected AND NOT "DB_Data".F13.Btt_Up_Selected AND NOT "DB_Data".F12.Btt_Down_Selected AND NOT "DB_Data".F12.Btt_Up_Selected AND NOT "DB_Data".F11.Btt_Down_Selected AND NOT "DB_Data".F11.Btt_Up_Selected AND NOT "DB_Data".F10.Btt_Down_Selected AND NOT "DB_Data".F10.Btt_Up_Selected AND NOT "DB_Data".F9.Btt_Down_Selected AND NOT "DB_Data".F9.Btt_Up_Selected AND NOT "DB_Data".F8.Btt_Down_Selected AND NOT "DB_Data".F8.Btt_Up_Selected AND NOT "DB_Data".F7.Btt_Down_Selected AND NOT "DB_Data".F7.Btt_Up_Selected AND NOT "DB_Data".F6.Btt_Down_Selected AND NOT "DB_Data".F6.Btt_Up_Selected AND NOT "DB_Data".F5.Btt_Down_Selected AND NOT "DB_Data".F5.Btt_Up_Selected AND NOT "DB_Data".F4.Btt_Down_Selected AND NOT "DB_Data".F4.Btt_Up_Selected AND NOT "DB_Data".F3.Btt_Down_Selected AND NOT "DB_Data".F3.Btt_Up_Selected AND NOT "DB_Data".F2.Btt_Down_Selected AND NOT "DB_Data".F2.Btt_Up_Selected AND NOT "DB_Data".F1.Btt_Up_Selected) OR ("DB_Data".F15.Sensor_Correct_Position AND NOT "DB_Data".F14.Btt_Down_Selected AND NOT "DB_Data".F14.Btt_Up_Selected AND NOT "DB_Data".F13.Btt_Down_Selected AND NOT "DB_Data".F13.Btt_Up_Selected AND NOT "DB_Data".F12.Btt_Down_Selected AND NOT "DB_Data".F12.Btt_Up_Selected AND NOT "DB_Data".F11.Btt_Down_Selected AND NOT "DB_Data".F11.Btt_Up_Selected AND NOT "DB_Data".F10.Btt_Down_Selected AND NOT "DB_Data".F10.Btt_Up_Selected AND NOT "DB_Data".F9.Btt_Down_Selected AND NOT "DB_Data".F9.Btt_Up_Selected AND NOT "DB_Data".F8.Btt_Down_Selected AND NOT "DB_Data".F8.Btt_Up_Selected AND NOT "DB_Data".F7.Btt_Down_Selected AND NOT "DB_Data".F7.Btt_Up_Selected AND NOT "DB_Data".F6.Btt_Down_Selected AND NOT "DB_Data".F6.Btt_Up_Selected AND NOT "DB_Data".F5.Btt_Down_Selected AND NOT "DB_Data".F5.Btt_Up_Selected AND NOT "DB_Data".F4.Btt_Down_Selected AND NOT "DB_Data".F4.Btt_Up_Selected AND NOT "DB_Data".F3.Btt_Down_Selected AND NOT "DB_Data".F3.Btt_Up_Selected AND NOT "DB_Data".F2.Btt_Down_Selected AND NOT "DB_Data".F2.Btt_Up_Selected AND NOT "DB_Data".F1.Btt_Up_Selected) OR ("DB_Data".F16.Sensor_Correct_Position AND NOT "DB_Data".F15.Btt_Down_Selected AND NOT "DB_Data".F15.Btt_Up_Selected AND NOT "DB_Data".F14.Btt_Down_Selected AND NOT "DB_Data".F14.Btt_Up_Selected AND NOT "DB_Data".F13.Btt_Down_Selected AND NOT "DB_Data".F13.Btt_Up_Selected AND NOT "DB_Data".F12.Btt_Down_Selected AND NOT "DB_Data".F12.Btt_Up_Selected AND NOT "DB_Data".F11.Btt_Down_Selected AND NOT "DB_Data".F11.Btt_Up_Selected AND NOT "DB_Data".F10.Btt_Down_Selected AND NOT "DB_Data".F10.Btt_Up_Selected AND NOT "DB_Data".F9.Btt_Down_Selected AND NOT "DB_Data".F9.Btt_Up_Selected AND NOT "DB_Data".F8.Btt_Down_Selected AND NOT "DB_Data".F8.Btt_Up_Selected AND NOT "DB_Data".F7.Btt_Down_Selected AND NOT "DB_Data".F7.Btt_Up_Selected AND NOT "DB_Data".F6.Btt_Down_Selected AND NOT "DB_Data".F6.Btt_Up_Selected AND NOT "DB_Data".F5.Btt_Down_Selected AND NOT "DB_Data".F5.Btt_Up_Selected AND NOT "DB_Data".F4.Btt_Down_Selected AND NOT "DB_Data".F4.Btt_Up_Selected AND NOT "DB_Data".F3.Btt_Down_Selected AND NOT "DB_Data".F3.Btt_Up_Selected AND NOT "DB_Data".F2.Btt_Down_Selected AND NOT "DB_Data".F2.Btt_Up_Selected AND NOT "DB_Data".F1.Btt_Up_Selected) OR ("DB_Data".F17.Sensor_Correct_Position AND NOT "DB_Data".F16.Btt_Down_Selected AND NOT "DB_Data".F16.Btt_Up_Selected AND NOT "DB_Data".F15.Btt_Down_Selected AND NOT "DB_Data".F15.Btt_Up_Selected AND NOT "DB_Data".F14.Btt_Down_Selected AND NOT "DB_Data".F14.Btt_Up_Selected AND NOT "DB_Data".F13.Btt_Down_Selected AND NOT "DB_Data".F13.Btt_Up_Selected AND NOT "DB_Data".F12.Btt_Down_Selected AND NOT "DB_Data".F12.Btt_Up_Selected AND NOT "DB_Data".F11.Btt_Down_Selected AND NOT "DB_Data".F11.Btt_Up_Selected AND NOT "DB_Data".F10.Btt_Down_Selected AND NOT "DB_Data".F10.Btt_Up_Selected AND NOT "DB_Data".F9.Btt_Down_Selected AND NOT "DB_Data".F9.Btt_Up_Selected AND NOT "DB_Data".F8.Btt_Down_Selected AND NOT "DB_Data".F8.Btt_Up_Selected AND NOT "DB_Data".F7.Btt_Down_Selected AND NOT "DB_Data".F7.Btt_Up_Selected AND NOT "DB_Data".F6.Btt_Down_Selected AND NOT "DB_Data".F6.Btt_Up_Selected AND NOT "DB_Data".F5.Btt_Down_Selected AND NOT "DB_Data".F5.Btt_Up_Selected AND NOT "DB_Data".F4.Btt_Down_Selected AND NOT "DB_Data".F4.Btt_Up_Selected AND NOT "DB_Data".F3.Btt_Down_Selected AND NOT "DB_Data".F3.Btt_Up_Selected AND NOT "DB_Data".F2.Btt_Down_Selected AND NOT "DB_Data".F2.Btt_Up_Selected AND NOT "DB_Data".F1.Btt_Up_Selected) OR ("DB_Data".F18.Sensor_Correct_Position AND NOT "DB_Data".F17.Btt_Down_Selected AND NOT "DB_Data".F17.Btt_Up_Selected AND NOT "DB_Data".F16.Btt_Down_Selected AND NOT "DB_Data".F16.Btt_Up_Selected AND NOT "DB_Data".F15.Btt_Down_Selected AND NOT "DB_Data".F15.Btt_Up_Selected AND NOT "DB_Data".F14.Btt_Down_Selected AND NOT "DB_Data".F14.Btt_Up_Selected AND NOT "DB_Data".F13.Btt_Down_Selected AND NOT "DB_Data".F13.Btt_Up_Selected AND NOT "DB_Data".F12.Btt_Down_Selected AND NOT "DB_Data".F12.Btt_Up_Selected AND NOT "DB_Data".F11.Btt_Down_Selected AND NOT "DB_Data".F11.Btt_Up_Selected AND NOT "DB_Data".F10.Btt_Down_Selected AND NOT "DB_Data".F10.Btt_Up_Selected AND NOT "DB_Data".F9.Btt_Down_Selected AND NOT "DB_Data".F9.Btt_Up_Selected AND NOT "DB_Data".F8.Btt_Down_Selected AND NOT "DB_Data".F8.Btt_Up_Selected AND NOT "DB_Data".F7.Btt_Down_Selected AND NOT "DB_Data".F7.Btt_Up_Selected AND NOT "DB_Data".F6.Btt_Down_Selected AND NOT "DB_Data".F6.Btt_Up_Selected AND NOT "DB_Data".F5.Btt_Down_Selected AND NOT "DB_Data".F5.Btt_Up_Selected AND NOT "DB_Data".F4.Btt_Down_Selected AND NOT "DB_Data".F4.Btt_Up_Selected AND NOT "DB_Data".F3.Btt_Down_Selected AND NOT "DB_Data".F3.Btt_Up_Selected AND NOT "DB_Data".F2.Btt_Down_Selected AND NOT "DB_Data".F2.Btt_Up_Selected AND NOT "DB_Data".F1.Btt_Up_Selected) OR ("DB_Data".F19.Sensor_Correct_Position AND NOT "DB_Data".F18.Btt_Down_Selected AND NOT "DB_Data".F18.Btt_Up_Selected AND NOT "DB_Data".F17.Btt_Down_Selected AND NOT "DB_Data".F17.Btt_Up_Selected AND NOT "DB_Data".F16.Btt_Down_Selected AND NOT "DB_Data".F16.Btt_Up_Selected AND NOT "DB_Data".F15.Btt_Down_Selected AND NOT "DB_Data".F15.Btt_Up_Selected AND NOT "DB_Data".F14.Btt_Down_Selected AND NOT "DB_Data".F14.Btt_Up_Selected AND NOT "DB_Data".F13.Btt_Down_Selected AND NOT "DB_Data".F13.Btt_Up_Selected AND NOT "DB_Data".F12.Btt_Down_Selected AND NOT "DB_Data".F12.Btt_Up_Selected AND NOT "DB_Data".F11.Btt_Down_Selected AND NOT "DB_Data".F11.Btt_Up_Selected AND NOT "DB_Data".F10.Btt_Down_Selected AND NOT "DB_Data".F10.Btt_Up_Selected AND NOT "DB_Data".F9.Btt_Down_Selected AND NOT "DB_Data".F9.Btt_Up_Selected AND NOT "DB_Data".F8.Btt_Down_Selected AND NOT "DB_Data".F8.Btt_Up_Selected AND NOT "DB_Data".F7.Btt_Down_Selected AND NOT "DB_Data".F7.Btt_Up_Selected AND NOT "DB_Data".F6.Btt_Down_Selected AND NOT "DB_Data".F6.Btt_Up_Selected AND NOT "DB_Data".F5.Btt_Down_Selected AND NOT "DB_Data".F5.Btt_Up_Selected AND NOT "DB_Data".F4.Btt_Down_Selected AND NOT "DB_Data".F4.Btt_Up_Selected AND NOT "DB_Data".F3.Btt_Down_Selected AND NOT "DB_Data".F3.Btt_Up_Selected AND NOT "DB_Data".F2.Btt_Down_Selected AND NOT "DB_Data".F2.Btt_Up_Selected AND NOT "DB_Data".F1.Btt_Up_Selected) OR ("DB_Data".F20.Sensor_Correct_Position AND NOT "DB_Data".F19.Btt_Down_Selected AND NOT "DB_Data".F19.Btt_Up_Selected AND NOT "DB_Data".F18.Btt_Down_Selected AND NOT "DB_Data".F18.Btt_Up_Selected AND NOT "DB_Data".F17.Btt_Down_Selected AND NOT "DB_Data".F17.Btt_Up_Selected AND NOT "DB_Data".F16.Btt_Down_Selected AND NOT "DB_Data".F16.Btt_Up_Selected AND NOT "DB_Data".F15.Btt_Down_Selected AND NOT "DB_Data".F15.Btt_Up_Selected AND NOT "DB_Data".F14.Btt_Down_Selected AND NOT "DB_Data".F14.Btt_Up_Selected AND NOT "DB_Data".F13.Btt_Down_Selected AND NOT "DB_Data".F13.Btt_Up_Selected AND NOT "DB_Data".F12.Btt_Down_Selected AND NOT "DB_Data".F12.Btt_Up_Selected AND NOT "DB_Data".F11.Btt_Down_Selected AND NOT "DB_Data".F11.Btt_Up_Selected AND NOT "DB_Data".F10.Btt_Down_Selected AND NOT "DB_Data".F10.Btt_Up_Selected AND NOT "DB_Data".F9.Btt_Down_Selected AND NOT "DB_Data".F9.Btt_Up_Selected AND NOT "DB_Data".F8.Btt_Down_Selected AND NOT "DB_Data".F8.Btt_Up_Selected AND NOT "DB_Data".F7.Btt_Down_Selected AND NOT "DB_Data".F7.Btt_Up_Selected AND NOT "DB_Data".F6.Btt_Down_Selected AND NOT "DB_Data".F6.Btt_Up_Selected AND NOT "DB_Data".F5.Btt_Down_Selected AND NOT "DB_Data".F5.Btt_Up_Selected AND NOT "DB_Data".F4.Btt_Down_Selected AND NOT "DB_Data".F4.Btt_Up_Selected AND NOT "DB_Data".F3.Btt_Down_Selected AND NOT "DB_Data".F3.Btt_Up_Selected AND NOT "DB_Data".F2.Btt_Down_Selected AND NOT "DB_Data".F2.Btt_Up_Selected AND NOT "DB_Data".F1.Btt_Up_Selected)) THEN
       "DB_Data".Last_Is_Down := FALSE;
   END_IF;
